Yaskawa INFORM job: DEMO_ROOF_SIDE_0625_3PAINT_61.JBI

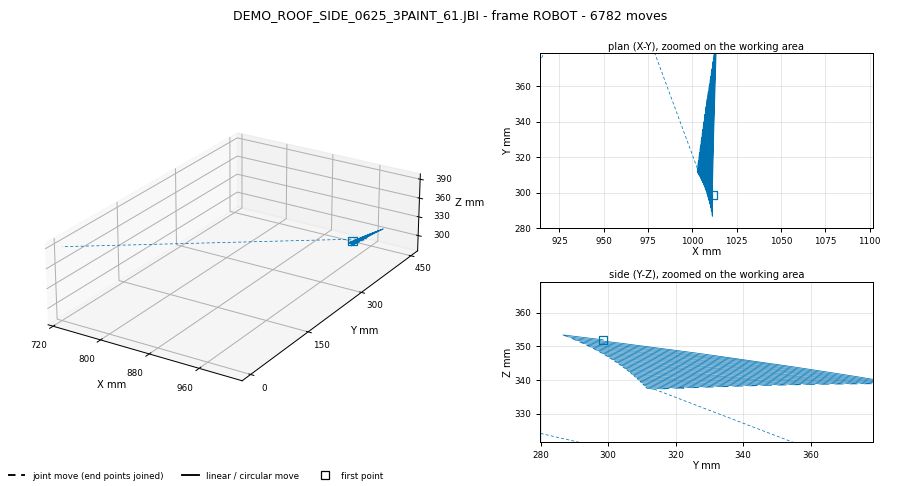
[picture p0: tool path of DEMO_ROOF_SIDE_0625_3PAINT_61.JBI in frame ROBOT, 6782 of 6782 moves have a stored position in this frame; points joined in program order, loops and branches not executed]
/JOB
//NAME DEMO_ROOF_SIDE_0625_3PAINT61
//POS
///NPOS 6782,0,0,0,0,0
///TOOL 0
///USER 0
///POSTYPE ROBOT
///RECTAN
///RCONF 1,0,0,0,0,0,0,0,0,0,0,0,0,0,0,0,0,0,0,0,0,0,0,0
C00000=1011.478,298.564,351.935,169.230,53.497,160.314
C00001=1011.473,298.316,351.966,169.223,53.504,160.314
C00002=1011.467,298.068,351.996,169.218,53.510,160.315
C00003=1011.462,297.820,352.027,169.211,53.517,160.315
C00004=1011.456,297.573,352.058,169.204,53.524,160.315
C00005=1011.451,297.324,352.089,169.198,53.530,160.315
C00006=1011.445,297.077,352.119,169.192,53.537,160.315
C00007=1011.440,296.828,352.150,169.186,53.544,160.316
C00008=1011.434,296.581,352.180,169.180,53.551,160.316
C00009=1011.429,296.332,352.211,169.174,53.558,160.316
C00010=1011.424,296.084,352.241,169.167,53.565,160.316
C00011=1011.418,295.836,352.272,169.161,53.572,160.317
C00012=1011.413,295.588,352.302,169.155,53.578,160.317
C00013=1011.408,295.340,352.333,169.148,53.585,160.317
C00014=1011.402,295.093,352.363,169.142,53.592,160.317
C00015=1011.398,294.844,352.393,169.136,53.599,160.317
C00016=1011.392,294.596,352.424,169.130,53.605,160.318
C00017=1011.387,294.348,352.455,169.123,53.612,160.318
C00018=1011.381,294.100,352.485,169.117,53.620,160.318
C00019=1011.376,293.852,352.515,169.111,53.626,160.319
C00020=1011.369,293.566,352.550,169.104,53.634,160.319
C00021=1011.364,293.280,352.585,169.097,53.642,160.319
C00022=1011.358,292.995,352.620,169.090,53.650,160.319
C00023=1011.352,292.709,352.655,169.082,53.658,160.320
C00024=1011.347,292.461,352.685,169.077,53.665,160.320
C00025=1011.341,292.212,352.715,169.070,53.672,160.320
C00026=1011.336,291.964,352.745,169.065,53.679,160.321
C00027=1011.331,291.716,352.775,169.058,53.686,160.321
C00028=1011.326,291.468,352.806,169.051,53.693,160.321
C00029=1011.320,291.220,352.835,169.046,53.700,160.321
C00030=1011.315,290.971,352.865,169.039,53.707,160.322
C00031=1011.309,290.724,352.895,169.034,53.714,160.322
C00032=1011.304,290.476,352.925,169.027,53.721,160.322
C00033=1011.298,290.227,352.954,169.021,53.728,160.322
C00034=1011.293,289.979,352.985,169.015,53.736,160.323
C00035=1011.288,289.732,353.014,169.009,53.742,160.323
C00036=1011.283,289.483,353.044,169.002,53.750,160.324
C00037=1011.277,289.235,353.074,168.997,53.757,160.324
C00038=1011.272,288.987,353.103,168.990,53.764,160.324
C00039=1011.267,288.739,353.133,168.985,53.771,160.324
C00040=1011.261,288.491,353.163,168.979,53.779,160.325
C00041=1011.256,288.243,353.192,168.972,53.785,160.325
C00042=1011.251,287.995,353.222,168.967,53.793,160.325
C00043=1011.245,287.746,353.251,168.960,53.800,160.326
C00044=1011.240,287.463,353.285,168.953,53.808,160.326
C00045=1011.233,287.181,353.318,168.946,53.816,160.326
C00046=1011.227,286.898,353.352,168.940,53.824,160.327
C00047=1011.221,286.616,353.386,168.933,53.833,160.327
C00048=1010.990,287.953,352.862,168.938,53.865,160.336
C00049=1010.994,288.177,352.835,168.944,53.858,160.335
C00050=1010.999,288.403,352.809,168.949,53.852,160.335
C00051=1011.004,288.627,352.782,168.955,53.845,160.335
C00052=1011.008,288.853,352.755,168.961,53.839,160.335
C00053=1011.014,289.077,352.728,168.965,53.832,160.334
C00054=1011.018,289.303,352.701,168.971,53.826,160.334
C00055=1011.023,289.527,352.674,168.977,53.819,160.334
C00056=1011.027,289.753,352.647,168.983,53.813,160.334
C00057=1011.033,290.001,352.618,168.989,53.806,160.333
C00058=1011.038,290.249,352.588,168.995,53.799,160.333
C00059=1011.043,290.497,352.558,169.001,53.792,160.333
C00060=1011.049,290.745,352.529,169.007,53.785,160.332
C00061=1011.054,290.993,352.499,169.013,53.778,160.332
C00062=1011.060,291.242,352.469,169.020,53.770,160.332
C00063=1011.064,291.489,352.439,169.025,53.764,160.332
C00064=1011.070,291.738,352.409,169.032,53.756,160.331
C00065=1011.075,291.986,352.379,169.038,53.749,160.331
C00066=1011.081,292.233,352.349,169.044,53.743,160.331
C00067=1011.085,292.482,352.319,169.051,53.736,160.331
C00068=1011.091,292.730,352.289,169.056,53.728,160.330
C00069=1011.096,293.018,352.254,169.063,53.720,160.330
C00070=1011.103,293.306,352.219,169.070,53.712,160.330
C00071=1011.110,293.594,352.183,169.078,53.704,160.329
C00072=1011.115,293.882,352.148,169.085,53.696,160.329
C00073=1011.121,294.130,352.118,169.092,53.689,160.329
C00074=1011.126,294.379,352.087,169.097,53.683,160.329
C00075=1011.131,294.627,352.057,169.104,53.676,160.328
C00076=1011.136,294.874,352.027,169.111,53.669,160.328
C00077=1011.141,295.122,351.997,169.117,53.662,160.328
C00078=1011.147,295.371,351.966,169.123,53.655,160.328
C00079=1011.152,295.618,351.936,169.128,53.648,160.327
C00080=1011.157,295.867,351.905,169.135,53.641,160.327
C00081=1011.163,296.115,351.875,169.141,53.635,160.327
C00082=1011.168,296.363,351.844,169.148,53.628,160.327
C00083=1011.174,296.611,351.814,169.154,53.621,160.327
C00084=1011.179,296.859,351.783,169.160,53.614,160.326
C00085=1011.185,297.107,351.752,169.167,53.607,160.326
C00086=1011.189,297.354,351.722,169.172,53.601,160.326
C00087=1011.195,297.603,351.692,169.179,53.594,160.326
C00088=1011.200,297.851,351.661,169.186,53.587,160.326
C00089=1011.205,298.099,351.630,169.192,53.581,160.325
C00090=1011.211,298.347,351.600,169.198,53.574,160.325
C00091=1011.216,298.595,351.569,169.204,53.567,160.325
C00092=1011.222,298.843,351.539,169.211,53.560,160.325
C00093=1011.227,299.091,351.508,169.218,53.554,160.325
C00094=1011.233,299.339,351.477,169.224,53.547,160.324
C00095=1011.238,299.588,351.446,169.230,53.540,160.324
C00096=1011.244,299.835,351.416,169.237,53.534,160.324
C00097=1011.249,300.084,351.385,169.243,53.527,160.324
C00098=1011.255,300.331,351.354,169.250,53.520,160.324
C00099=1011.260,300.580,351.324,169.255,53.514,160.323
C00100=1011.266,300.827,351.293,169.262,53.507,160.323
C00101=1011.271,301.075,351.262,169.269,53.500,160.323
C00102=1011.277,301.323,351.231,169.275,53.494,160.323
C00103=1011.282,301.571,351.200,169.282,53.487,160.323
C00104=1011.288,301.819,351.169,169.287,53.480,160.323
C00105=1011.294,302.067,351.139,169.295,53.474,160.323
C00106=1011.299,302.315,351.108,169.301,53.467,160.322
C00107=1011.304,302.563,351.077,169.307,53.461,160.322
C00108=1011.311,302.811,351.046,169.314,53.454,160.322
C00109=1011.316,303.059,351.015,169.321,53.448,160.322
C00110=1011.322,303.307,350.985,169.327,53.441,160.322
C00111=1011.327,303.555,350.954,169.333,53.434,160.322
C00112=1011.333,303.803,350.923,169.340,53.428,160.322
C00113=1011.338,304.051,350.892,169.346,53.422,160.321
C00114=1011.345,304.299,350.861,169.353,53.415,160.321
C00115=1011.350,304.547,350.829,169.359,53.409,160.321
C00116=1011.356,304.795,350.799,169.366,53.402,160.321
C00117=1011.362,305.043,350.767,169.373,53.395,160.321
C00118=1011.368,305.291,350.736,169.379,53.389,160.321
C00119=1011.373,305.539,350.706,169.386,53.382,160.321
C00120=1011.380,305.787,350.674,169.393,53.376,160.321
C00121=1011.385,306.035,350.643,169.398,53.370,160.320
C00122=1011.391,306.282,350.612,169.405,53.363,160.320
C00123=1011.396,306.531,350.581,169.412,53.356,160.320
C00124=1011.403,306.778,350.550,169.418,53.350,160.320
C00125=1011.408,307.026,350.519,169.425,53.344,160.320
C00126=1011.414,307.274,350.487,169.432,53.337,160.320
C00127=1011.419,307.522,350.456,169.438,53.331,160.320
C00128=1011.425,307.770,350.424,169.445,53.325,160.320
C00129=1011.433,308.076,350.386,169.454,53.316,160.320
C00130=1011.440,308.383,350.348,169.461,53.309,160.320
C00131=1011.448,308.689,350.309,169.470,53.301,160.319
C00132=1011.455,308.995,350.270,169.479,53.293,160.319
C00133=1011.460,309.243,350.238,169.484,53.287,160.319
C00134=1011.465,309.491,350.206,169.491,53.281,160.319
C00135=1011.471,309.739,350.174,169.498,53.275,160.319
C00136=1011.476,309.986,350.142,169.505,53.269,160.319
C00137=1011.482,310.235,350.110,169.511,53.263,160.319
C00138=1011.488,310.481,350.078,169.518,53.256,160.319
C00139=1011.494,310.730,350.046,169.525,53.250,160.319
C00140=1011.498,310.977,350.014,169.531,53.244,160.319
C00141=1011.504,311.226,349.981,169.538,53.238,160.319
C00142=1011.510,311.473,349.950,169.545,53.232,160.319
C00143=1011.516,311.721,349.918,169.551,53.225,160.319
C00144=1011.521,311.969,349.886,169.559,53.219,160.319
C00145=1011.528,312.216,349.853,169.565,53.213,160.319
C00146=1011.533,312.464,349.822,169.572,53.207,160.319
C00147=1011.538,312.713,349.789,169.578,53.201,160.319
C00148=1011.544,312.961,349.757,169.585,53.195,160.319
C00149=1011.550,313.208,349.725,169.592,53.189,160.319
C00150=1011.556,313.456,349.693,169.599,53.183,160.319
C00151=1011.561,313.703,349.661,169.606,53.177,160.319
C00152=1011.567,313.951,349.628,169.612,53.171,160.319
C00153=1011.573,314.199,349.596,169.619,53.165,160.319
C00154=1011.578,314.447,349.564,169.627,53.158,160.319
C00155=1011.584,314.695,349.531,169.633,53.153,160.319
C00156=1011.590,314.943,349.499,169.640,53.146,160.319
C00157=1011.597,315.190,349.466,169.646,53.141,160.319
C00158=1011.601,315.438,349.434,169.653,53.134,160.319
C00159=1011.608,315.686,349.401,169.661,53.128,160.319
C00160=1011.614,315.934,349.369,169.667,53.123,160.319
C00161=1011.620,316.182,349.337,169.674,53.116,160.319
C00162=1011.625,316.429,349.305,169.681,53.110,160.319
C00163=1011.632,316.677,349.272,169.688,53.105,160.319
C00164=1011.637,316.925,349.240,169.695,53.099,160.319
C00165=1011.643,317.173,349.207,169.701,53.093,160.319
C00166=1011.649,317.421,349.175,169.709,53.087,160.319
C00167=1011.655,317.668,349.143,169.716,53.081,160.319
C00168=1011.661,317.916,349.110,169.722,53.076,160.319
C00169=1011.667,318.164,349.078,169.730,53.069,160.319
C00170=1011.673,318.412,349.044,169.737,53.063,160.319
C00171=1011.679,318.659,349.012,169.743,53.057,160.319
C00172=1011.685,318.907,348.980,169.751,53.052,160.319
C00173=1011.691,319.155,348.947,169.758,53.046,160.320
C00174=1011.698,319.403,348.914,169.764,53.040,160.319
C00175=1011.703,319.651,348.882,169.771,53.034,160.319
C00176=1011.709,319.899,348.849,169.779,53.028,160.320
C00177=1011.715,320.146,348.816,169.785,53.023,160.320
C00178=1011.722,320.394,348.783,169.792,53.016,160.320
C00179=1011.728,320.642,348.751,169.800,53.011,160.320
C00180=1011.734,320.889,348.718,169.806,53.005,160.320
C00181=1011.739,321.138,348.685,169.814,53.000,160.320
C00182=1011.746,321.385,348.652,169.821,52.994,160.320
C00183=1011.752,321.633,348.620,169.827,52.988,160.320
C00184=1011.758,321.880,348.587,169.835,52.982,160.320
C00185=1011.765,322.128,348.554,169.842,52.976,160.320
C00186=1011.770,322.376,348.521,169.849,52.971,160.321
C00187=1011.777,322.624,348.488,169.856,52.965,160.321
C00188=1011.783,322.871,348.455,169.864,52.959,160.321
C00189=1011.791,323.183,348.414,169.873,52.952,160.321
C00190=1011.799,323.495,348.373,169.882,52.945,160.321
C00191=1011.807,323.807,348.331,169.891,52.938,160.321
C00192=1011.815,324.119,348.289,169.900,52.931,160.322
C00193=1011.821,324.366,348.257,169.906,52.925,160.321
C00194=1011.827,324.614,348.224,169.914,52.920,160.322
C00195=1011.833,324.862,348.190,169.921,52.914,160.322
C00196=1011.839,325.109,348.158,169.929,52.908,160.322
C00197=1011.847,325.357,348.124,169.936,52.903,160.322
C00198=1011.853,325.604,348.091,169.943,52.897,160.322
C00199=1011.859,325.852,348.057,169.951,52.891,160.322
C00200=1011.864,326.100,348.024,169.957,52.886,160.323
C00201=1011.871,326.347,347.990,169.965,52.881,160.323
C00202=1011.877,326.595,347.957,169.973,52.875,160.323
C00203=1011.883,326.843,347.923,169.979,52.870,160.323
C00204=1011.889,327.090,347.890,169.986,52.864,160.323
C00205=1011.896,327.338,347.855,169.994,52.859,160.324
C00206=1011.901,327.586,347.822,170.001,52.854,160.324
C00207=1011.908,327.833,347.789,170.008,52.848,160.324
C00208=1011.914,328.081,347.754,170.016,52.843,160.324
C00209=1011.920,328.329,347.721,170.023,52.838,160.324
C00210=1011.926,328.576,347.687,170.030,52.832,160.325
C00211=1011.933,328.824,347.653,170.038,52.827,160.325
C00212=1011.939,329.071,347.620,170.046,52.821,160.325
C00213=1011.946,329.319,347.586,170.052,52.816,160.325
C00214=1011.951,329.567,347.552,170.060,52.811,160.325
C00215=1011.958,329.814,347.519,170.068,52.805,160.326
C00216=1011.964,330.062,347.485,170.074,52.800,160.326
C00217=1011.970,330.310,347.450,170.082,52.795,160.326
C00218=1011.977,330.557,347.417,170.090,52.789,160.326
C00219=1011.983,330.804,347.383,170.097,52.784,160.327
C00220=1011.990,331.052,347.348,170.104,52.778,160.327
C00221=1011.996,331.299,347.315,170.112,52.773,160.327
C00222=1012.002,331.548,347.281,170.119,52.768,160.327
C00223=1012.008,331.795,347.247,170.127,52.762,160.327
C00224=1012.016,332.042,347.212,170.134,52.757,160.328
C00225=1012.022,332.290,347.178,170.142,52.752,160.328
C00226=1012.028,332.538,347.144,170.150,52.747,160.328
C00227=1012.034,332.786,347.110,170.156,52.742,160.328
C00228=1012.040,333.033,347.076,170.164,52.736,160.329
C00229=1012.047,333.281,347.041,170.172,52.731,160.329
C00230=1012.053,333.528,347.007,170.180,52.726,160.329
C00231=1012.059,333.776,346.972,170.186,52.721,160.330
C00232=1012.066,334.024,346.937,170.194,52.716,160.330
C00233=1012.072,334.271,346.903,170.202,52.711,160.330
C00234=1012.079,334.519,346.870,170.210,52.705,160.330
C00235=1012.086,334.766,346.834,170.217,52.701,160.331
C00236=1012.092,335.013,346.800,170.225,52.695,160.331
C00237=1012.098,335.261,346.766,170.233,52.691,160.332
C00238=1012.105,335.509,346.731,170.240,52.685,160.332
C00239=1012.111,335.756,346.697,170.248,52.681,160.332
C00240=1012.117,336.003,346.662,170.255,52.675,160.332
C00241=1012.124,336.251,346.627,170.263,52.670,160.333
C00242=1012.130,336.499,346.593,170.271,52.665,160.333
C00243=1012.137,336.746,346.558,170.278,52.661,160.333
C00244=1012.144,336.993,346.524,170.286,52.655,160.334
C00245=1012.150,337.241,346.489,170.294,52.650,160.334
C00246=1012.157,337.489,346.455,170.302,52.645,160.334
C00247=1012.164,337.736,346.420,170.310,52.640,160.335
C00248=1012.170,337.984,346.384,170.316,52.635,160.335
C00249=1012.178,338.291,346.342,170.326,52.629,160.335
C00250=1012.186,338.599,346.298,170.336,52.623,160.336
C00251=1012.194,338.907,346.255,170.346,52.617,160.337
C00252=1012.202,339.213,346.211,170.355,52.611,160.337
C00253=1012.209,339.461,346.176,170.364,52.606,160.337
C00254=1012.216,339.708,346.141,170.371,52.601,160.338
C00255=1012.223,339.956,346.106,170.378,52.596,160.338
C00256=1012.229,340.203,346.070,170.386,52.591,160.338
C00257=1012.235,340.451,346.035,170.395,52.587,160.339
C00258=1012.242,340.699,346.000,170.403,52.582,160.339
C00259=1012.249,340.946,345.965,170.410,52.576,160.340
C00260=1012.255,341.193,345.930,170.418,52.572,160.340
C00261=1012.262,341.441,345.895,170.426,52.567,160.340
C00262=1012.268,341.688,345.859,170.434,52.562,160.341
C00263=1012.275,341.935,345.823,170.442,52.558,160.341
C00264=1012.282,342.182,345.788,170.450,52.553,160.342
C00265=1012.289,342.430,345.753,170.458,52.548,160.342
C00266=1012.296,342.677,345.718,170.465,52.544,160.343
C00267=1012.302,342.925,345.682,170.473,52.539,160.343
C00268=1012.309,343.173,345.647,170.481,52.534,160.344
C00269=1012.316,343.420,345.611,170.490,52.529,160.344
C00270=1012.323,343.667,345.576,170.498,52.525,160.344
C00271=1012.329,343.915,345.540,170.506,52.520,160.345
C00272=1012.336,344.162,345.505,170.514,52.515,160.345
C00273=1012.343,344.409,345.469,170.521,52.511,160.346
C00274=1012.350,344.657,345.434,170.530,52.506,160.346
C00275=1012.356,344.905,345.398,170.538,52.502,160.347
C00276=1012.363,345.151,345.362,170.546,52.497,160.347
C00277=1012.370,345.399,345.327,170.554,52.492,160.348
C00278=1012.378,345.646,345.291,170.562,52.487,160.348
C00279=1012.384,345.894,345.255,170.571,52.483,160.349
C00280=1012.391,346.141,345.219,170.579,52.478,160.349
C00281=1012.397,346.388,345.184,170.587,52.474,160.350
C00282=1012.404,346.636,345.147,170.594,52.469,160.350
C00283=1012.411,346.883,345.112,170.602,52.465,160.351
C00284=1012.417,347.130,345.076,170.611,52.460,160.351
C00285=1012.425,347.378,345.039,170.619,52.456,160.352
C00286=1012.431,347.625,345.004,170.627,52.451,160.352
C00287=1012.438,347.872,344.968,170.635,52.447,160.353
C00288=1012.445,348.120,344.931,170.644,52.443,160.353
C00289=1012.452,348.366,344.895,170.652,52.438,160.354
C00290=1012.459,348.614,344.858,170.661,52.434,160.355
C00291=1012.466,348.862,344.823,170.669,52.429,160.355
C00292=1012.472,349.109,344.787,170.676,52.425,160.356
C00293=1012.480,349.356,344.750,170.684,52.420,160.356
C00294=1012.486,349.603,344.714,170.693,52.416,160.357
C00295=1012.494,349.851,344.678,170.701,52.412,160.357
C00296=1012.500,350.098,344.641,170.710,52.407,160.358
C00297=1012.508,350.345,344.605,170.718,52.403,160.358
C00298=1012.514,350.592,344.569,170.726,52.399,160.359
C00299=1012.522,350.840,344.532,170.735,52.394,160.360
C00300=1012.528,351.087,344.496,170.743,52.390,160.360
C00301=1012.536,351.334,344.460,170.751,52.386,160.361
C00302=1012.543,351.582,344.423,170.760,52.381,160.361
C00303=1012.550,351.828,344.386,170.768,52.377,160.362
C00304=1012.557,352.076,344.350,170.777,52.373,160.362
C00305=1012.564,352.322,344.314,170.785,52.368,160.363
C00306=1012.571,352.570,344.277,170.794,52.364,160.364
C00307=1012.579,352.818,344.241,170.802,52.360,160.364
C00308=1012.586,353.064,344.204,170.810,52.355,160.365
C00309=1012.594,353.369,344.158,170.821,52.351,160.366
C00310=1012.603,353.675,344.113,170.832,52.346,160.367
C00311=1012.612,353.979,344.068,170.842,52.340,160.367
C00312=1012.621,354.284,344.022,170.852,52.335,160.368
C00313=1012.628,354.531,343.985,170.861,52.331,160.369
C00314=1012.634,354.778,343.948,170.869,52.327,160.369
C00315=1012.642,355.025,343.911,170.879,52.322,160.370
C00316=1012.649,355.273,343.875,170.887,52.318,160.371
C00317=1012.657,355.520,343.837,170.896,52.314,160.371
C00318=1012.665,355.767,343.800,170.904,52.310,160.372
C00319=1012.671,356.014,343.764,170.913,52.306,160.373
C00320=1012.678,356.261,343.726,170.922,52.302,160.373
C00321=1012.685,356.508,343.689,170.930,52.298,160.374
C00322=1012.693,356.756,343.652,170.939,52.294,160.375
C00323=1012.700,357.003,343.615,170.948,52.290,160.376
C00324=1012.708,357.250,343.577,170.956,52.286,160.376
C00325=1012.715,357.497,343.540,170.965,52.282,160.377
C00326=1012.723,357.744,343.503,170.973,52.278,160.378
C00327=1012.730,357.992,343.466,170.982,52.274,160.378
C00328=1012.737,358.239,343.429,170.991,52.270,160.379
C00329=1012.744,358.486,343.391,171.000,52.266,160.380
C00330=1012.752,358.733,343.353,171.009,52.262,160.381
C00331=1012.758,358.979,343.316,171.018,52.258,160.381
C00332=1012.766,359.226,343.278,171.026,52.254,160.382
C00333=1012.773,359.473,343.241,171.035,52.251,160.383
C00334=1012.781,359.721,343.203,171.044,52.247,160.384
C00335=1012.788,359.968,343.165,171.053,52.243,160.384
C00336=1012.795,360.215,343.128,171.061,52.239,160.385
C00337=1012.803,360.462,343.089,171.070,52.235,160.386
C00338=1012.810,360.709,343.052,171.080,52.231,160.387
C00339=1012.817,360.956,343.014,171.089,52.227,160.388
C00340=1012.825,361.203,342.976,171.098,52.224,160.389
C00341=1012.832,361.450,342.939,171.106,52.220,160.389
C00342=1012.839,361.697,342.901,171.115,52.216,160.390
C00343=1012.847,361.943,342.863,171.124,52.212,160.391
C00344=1012.855,362.191,342.825,171.134,52.208,160.392
C00345=1012.862,362.438,342.787,171.143,52.205,160.393
C00346=1012.870,362.685,342.749,171.151,52.201,160.393
C00347=1012.877,362.931,342.711,171.160,52.197,160.394
C00348=1012.885,363.179,342.673,171.169,52.194,160.395
C00349=1012.892,363.426,342.635,171.179,52.190,160.396
C00350=1012.900,363.673,342.597,171.188,52.186,160.397
C00351=1012.907,363.919,342.559,171.197,52.183,160.397
C00352=1012.915,364.167,342.520,171.206,52.179,160.398
C00353=1012.923,364.414,342.483,171.216,52.175,160.399
C00354=1012.930,364.660,342.445,171.225,52.172,160.400
C00355=1012.938,364.907,342.406,171.234,52.168,160.401
C00356=1012.946,365.155,342.368,171.243,52.165,160.402
C00357=1012.954,365.402,342.330,171.253,52.161,160.403
C00358=1012.961,365.648,342.292,171.262,52.157,160.404
C00359=1012.969,365.895,342.253,171.271,52.154,160.405
C00360=1012.977,366.142,342.215,171.280,52.151,160.405
C00361=1012.985,366.389,342.176,171.290,52.147,160.406
C00362=1012.993,366.636,342.138,171.299,52.143,160.407
C00363=1013.000,366.883,342.099,171.308,52.140,160.408
C00364=1013.008,367.130,342.060,171.318,52.136,160.409
C00365=1013.015,367.376,342.022,171.327,52.132,160.410
C00366=1013.023,367.624,341.983,171.336,52.129,160.411
C00367=1013.030,367.870,341.945,171.346,52.126,160.412
C00368=1013.039,368.117,341.905,171.355,52.122,160.413
C00369=1013.048,368.429,341.856,171.367,52.118,160.414
C00370=1013.057,368.742,341.807,171.379,52.114,160.415
C00371=1013.067,369.055,341.758,171.390,52.109,160.416
C00372=1013.077,369.367,341.709,171.403,52.105,160.418
C00373=1013.085,369.614,341.669,171.413,52.102,160.419
C00374=1013.093,369.860,341.631,171.422,52.098,160.420
C00375=1013.101,370.107,341.591,171.431,52.095,160.421
C00376=1013.108,370.355,341.552,171.441,52.091,160.422
C00377=1013.117,370.601,341.513,171.450,52.089,160.423
C00378=1013.124,370.848,341.475,171.460,52.085,160.424
C00379=1013.132,371.095,341.435,171.470,52.082,160.425
C00380=1013.140,371.342,341.396,171.479,52.078,160.426
C00381=1013.149,371.588,341.357,171.489,52.075,160.427
C00382=1013.156,371.835,341.317,171.498,52.072,160.428
C00383=1013.164,372.082,341.279,171.508,52.068,160.429
C00384=1013.172,372.329,341.239,171.518,52.066,160.430
C00385=1013.180,372.575,341.199,171.528,52.062,160.431
C00386=1013.189,372.822,341.160,171.537,52.059,160.432
C00387=1013.196,373.069,341.121,171.548,52.056,160.433
C00388=1013.205,373.316,341.082,171.557,52.053,160.434
C00389=1013.212,373.562,341.043,171.567,52.049,160.435
C00390=1013.220,373.809,341.003,171.576,52.046,160.436
C00391=1013.229,374.055,340.963,171.587,52.043,160.438
C00392=1013.237,374.302,340.924,171.596,52.040,160.439
C00393=1013.245,374.549,340.884,171.606,52.037,160.440
C00394=1013.253,374.796,340.845,171.616,52.034,160.441
C00395=1013.262,375.042,340.805,171.626,52.031,160.442
C00396=1013.269,375.289,340.766,171.636,52.028,160.443
C00397=1013.277,375.536,340.726,171.646,52.025,160.444
C00398=1013.285,375.782,340.685,171.655,52.022,160.445
C00399=1013.294,376.030,340.645,171.666,52.019,160.447
C00400=1013.302,376.276,340.605,171.676,52.015,160.448
C00401=1013.310,376.523,340.565,171.686,52.013,160.449
C00402=1013.318,376.769,340.525,171.696,52.009,160.450
C00403=1013.326,377.016,340.485,171.705,52.007,160.451
C00404=1013.334,377.263,340.445,171.716,52.004,160.453
C00405=1013.343,377.508,340.405,171.727,52.001,160.454
C00406=1013.351,377.755,340.365,171.736,51.998,160.455
C00407=1013.359,378.002,340.324,171.746,51.995,160.456
C00408=1013.368,378.249,340.285,171.756,51.992,160.457
C00409=1013.376,378.495,340.244,171.767,51.989,160.458
C00410=1013.384,378.742,340.203,171.777,51.986,160.460
C00411=1013.392,378.988,340.163,171.787,51.984,160.461
C00412=1013.401,379.235,340.123,171.797,51.980,160.462
C00413=1013.409,379.481,340.082,171.808,51.978,160.463
C00414=1013.417,379.728,340.042,171.817,51.975,160.465
C00415=1013.426,379.975,340.002,171.828,51.972,160.466
C00416=1013.434,380.221,339.961,171.839,51.969,160.467
C00417=1013.442,380.468,339.921,171.849,51.967,160.468
C00418=1013.451,380.714,339.880,171.859,51.964,160.470
C00419=1013.459,380.961,339.840,171.870,51.961,160.471
C00420=1013.468,381.207,339.799,171.880,51.958,160.472
C00421=1013.477,381.453,339.759,171.891,51.955,160.473
C00422=1013.485,381.700,339.718,171.901,51.953,160.475
C00423=1013.493,381.947,339.677,171.911,51.950,160.476
C00424=1013.503,382.193,339.637,171.922,51.947,160.477
C00425=1013.511,382.440,339.596,171.933,51.945,160.479
C00426=1013.520,382.687,339.555,171.943,51.942,160.480
C00427=1013.528,382.933,339.515,171.954,51.939,160.481
C00428=1013.537,383.179,339.473,171.964,51.936,160.483
C00429=1013.548,383.480,339.423,171.977,51.934,160.484
C00430=1013.558,383.781,339.373,171.990,51.930,160.486
C00431=1013.569,384.083,339.323,172.003,51.927,160.488
C00432=1013.580,384.384,339.273,172.017,51.924,160.489
C00433=1013.588,384.631,339.232,172.027,51.921,160.491
C00434=1013.597,384.877,339.191,172.037,51.919,160.492
C00435=1013.606,385.124,339.150,172.048,51.916,160.494
C00436=1013.615,385.370,339.108,172.059,51.914,160.495
C00437=1013.623,385.616,339.067,172.070,51.911,160.496
C00438=1013.632,385.863,339.026,172.080,51.908,160.498
C00439=1013.640,386.109,338.984,172.092,51.906,160.499
C00440=1013.649,386.356,338.942,172.103,51.904,160.501
C00441=1013.305,384.294,338.940,171.994,51.982,160.501
C00442=1013.295,384.035,338.983,171.984,51.985,160.499
C00443=1013.286,383.776,339.026,171.972,51.988,160.498
C00444=1013.277,383.517,339.069,171.961,51.991,160.496
C00445=1013.268,383.257,339.113,171.949,51.994,160.495
C00446=1013.259,383.011,339.153,171.939,51.996,160.494
C00447=1013.250,382.764,339.194,171.929,51.999,160.492
C00448=1013.242,382.518,339.235,171.918,52.001,160.491
C00449=1013.233,382.271,339.275,171.907,52.005,160.490
C00450=1013.225,382.025,339.316,171.897,52.007,160.488
C00451=1013.216,381.778,339.357,171.886,52.010,160.487
C00452=1013.208,381.532,339.397,171.875,52.013,160.486
C00453=1013.200,381.285,339.437,171.865,52.015,160.484
C00454=1013.191,381.038,339.478,171.855,52.018,160.483
C00455=1013.182,380.792,339.518,171.844,52.021,160.482
C00456=1013.174,380.545,339.559,171.833,52.024,160.480
C00457=1013.165,380.299,339.600,171.824,52.027,160.479
C00458=1013.157,380.053,339.640,171.813,52.029,160.478
C00459=1013.148,379.806,339.680,171.803,52.032,160.477
C00460=1013.140,379.559,339.721,171.792,52.035,160.475
C00461=1013.132,379.313,339.761,171.783,52.038,160.474
C00462=1013.123,379.066,339.802,171.772,52.041,160.473
C00463=1013.115,378.819,339.842,171.761,52.044,160.472
C00464=1013.107,378.573,339.882,171.751,52.047,160.470
C00465=1013.099,378.326,339.922,171.742,52.050,160.469
C00466=1013.090,378.079,339.963,171.731,52.052,160.468
C00467=1013.082,377.833,340.002,171.721,52.056,160.467
C00468=1013.074,377.587,340.043,171.711,52.059,160.466
C00469=1013.066,377.340,340.083,171.701,52.062,160.465
C00470=1013.058,377.093,340.124,171.690,52.064,160.463
C00471=1013.049,376.847,340.163,171.680,52.067,160.462
C00472=1013.041,376.601,340.203,171.670,52.071,160.461
C00473=1013.034,376.354,340.243,171.661,52.073,160.460
C00474=1013.025,376.107,340.283,171.650,52.077,160.459
C00475=1013.017,375.861,340.323,171.640,52.080,160.457
C00476=1013.009,375.613,340.364,171.631,52.083,160.456
C00477=1013.001,375.367,340.403,171.620,52.086,160.455
C00478=1012.993,375.120,340.443,171.611,52.089,160.454
C00479=1012.985,374.874,340.483,171.600,52.092,160.453
C00480=1012.977,374.627,340.522,171.591,52.095,160.452
C00481=1012.969,374.380,340.561,171.581,52.098,160.451
C00482=1012.961,374.133,340.601,171.570,52.101,160.449
C00483=1012.953,373.887,340.640,171.561,52.104,160.448
C00484=1012.944,373.640,340.680,171.551,52.108,160.447
C00485=1012.936,373.393,340.720,171.541,52.111,160.446
C00486=1012.928,373.147,340.759,171.531,52.114,160.445
C00487=1012.919,372.900,340.798,171.522,52.117,160.444
C00488=1012.912,372.653,340.837,171.512,52.121,160.443
C00489=1012.904,372.406,340.877,171.502,52.124,160.442
C00490=1012.895,372.159,340.916,171.492,52.128,160.441
C00491=1012.888,371.913,340.955,171.483,52.130,160.440
C00492=1012.880,371.666,340.994,171.473,52.134,160.439
C00493=1012.872,371.419,341.034,171.464,52.137,160.438
C00494=1012.864,371.172,341.073,171.453,52.140,160.437
C00495=1012.856,370.926,341.112,171.444,52.144,160.436
C00496=1012.849,370.678,341.151,171.434,52.147,160.435
C00497=1012.840,370.432,341.190,171.425,52.151,160.434
C00498=1012.833,370.185,341.228,171.414,52.154,160.433
C00499=1012.825,369.938,341.268,171.405,52.157,160.432
C00500=1012.817,369.691,341.307,171.396,52.160,160.431
C00501=1012.809,369.445,341.346,171.386,52.164,160.430
C00502=1012.799,369.130,341.396,171.374,52.169,160.429
C00503=1012.789,368.815,341.445,171.362,52.173,160.427
C00504=1012.779,368.500,341.495,171.350,52.177,160.426
C00505=1012.770,368.186,341.545,171.338,52.182,160.425
C00506=1012.762,367.939,341.583,171.328,52.185,160.424
C00507=1012.754,367.692,341.622,171.319,52.188,160.423
C00508=1012.747,367.445,341.661,171.309,52.192,160.422
C00509=1012.739,367.198,341.699,171.300,52.196,160.421
C00510=1012.731,366.951,341.737,171.292,52.199,160.420
C00511=1012.724,366.704,341.777,171.281,52.202,160.419
C00512=1012.717,366.457,341.815,171.272,52.206,160.418
C00513=1012.709,366.211,341.853,171.263,52.209,160.417
C00514=1012.701,365.964,341.892,171.253,52.213,160.416
C00515=1012.693,365.717,341.930,171.244,52.217,160.415
C00516=1012.685,365.470,341.969,171.236,52.221,160.415
C00517=1012.678,365.223,342.006,171.226,52.225,160.414
C00518=1012.670,364.976,342.045,171.217,52.228,160.413
C00519=1012.662,364.729,342.083,171.208,52.232,160.412
C00520=1012.655,364.482,342.120,171.198,52.235,160.411
C00521=1012.647,364.235,342.159,171.189,52.239,160.410
C00522=1012.639,363.988,342.197,171.180,52.242,160.409
C00523=1012.632,363.741,342.235,171.171,52.246,160.408
C00524=1012.624,363.495,342.273,171.161,52.250,160.408
C00525=1012.617,363.247,342.311,171.152,52.254,160.407
C00526=1012.609,363.000,342.349,171.143,52.257,160.406
C00527=1012.602,362.753,342.387,171.134,52.261,160.405
C00528=1012.594,362.507,342.425,171.125,52.265,160.404
C00529=1012.587,362.259,342.463,171.116,52.269,160.403
C00530=1012.579,362.012,342.501,171.107,52.272,160.402
C00531=1012.572,361.765,342.539,171.098,52.276,160.402
C00532=1012.564,361.518,342.576,171.088,52.280,160.401
C00533=1012.557,361.271,342.614,171.080,52.284,160.400
C00534=1012.550,361.024,342.652,171.071,52.288,160.399
C00535=1012.542,360.777,342.689,171.062,52.292,160.399
C00536=1012.535,360.531,342.728,171.053,52.295,160.398
C00537=1012.528,360.283,342.765,171.045,52.300,160.397
C00538=1012.520,360.036,342.803,171.035,52.303,160.396
C00539=1012.513,359.789,342.840,171.026,52.308,160.395
C00540=1012.506,359.542,342.878,171.017,52.311,160.395
C00541=1012.499,359.295,342.915,171.009,52.315,160.394
C00542=1012.491,359.048,342.954,171.000,52.319,160.393
C00543=1012.484,358.801,342.991,170.991,52.323,160.392
C00544=1012.477,358.554,343.029,170.982,52.327,160.392
C00545=1012.469,358.307,343.066,170.973,52.331,160.391
C00546=1012.462,358.059,343.103,170.964,52.335,160.390
C00547=1012.455,357.812,343.141,170.956,52.339,160.389
C00548=1012.448,357.565,343.178,170.947,52.343,160.389
C00549=1012.440,357.318,343.215,170.938,52.347,160.388
C00550=1012.433,357.071,343.253,170.930,52.351,160.387
C00551=1012.426,356.823,343.289,170.921,52.355,160.387
C00552=1012.418,356.576,343.327,170.911,52.359,160.386
C00553=1012.411,356.330,343.363,170.903,52.363,160.385
C00554=1012.404,356.082,343.400,170.894,52.368,160.384
C00555=1012.397,355.835,343.438,170.886,52.372,160.384
C00556=1012.390,355.588,343.475,170.877,52.376,160.383
C00557=1012.382,355.341,343.511,170.869,52.380,160.382
C00558=1012.375,355.094,343.549,170.860,52.384,160.382
C00559=1012.368,354.846,343.585,170.852,52.388,160.381
C00560=1012.360,354.600,343.622,170.843,52.392,160.380
C00561=1012.353,354.352,343.659,170.835,52.396,160.380
C00562=1012.345,354.045,343.705,170.823,52.402,160.379
C00563=1012.336,353.738,343.751,170.812,52.407,160.378
C00564=1012.327,353.430,343.796,170.802,52.412,160.377
C00565=1012.319,353.124,343.842,170.792,52.417,160.376
C00566=1012.311,352.876,343.878,170.783,52.421,160.376
C00567=1012.304,352.630,343.916,170.775,52.425,160.375
C00568=1012.298,352.382,343.952,170.767,52.430,160.375
C00569=1012.290,352.135,343.989,170.758,52.434,160.374
C00570=1012.283,351.888,344.025,170.749,52.438,160.373
C00571=1012.276,351.640,344.061,170.741,52.443,160.373
C00572=1012.269,351.393,344.098,170.733,52.447,160.372
C00573=1012.262,351.146,344.134,170.724,52.451,160.372
C00574=1012.255,350.899,344.170,170.716,52.456,160.371
C00575=1012.248,350.651,344.207,170.708,52.460,160.370
C00576=1012.241,350.404,344.243,170.699,52.464,160.370
C00577=1012.234,350.157,344.279,170.691,52.469,160.369
C00578=1012.227,349.910,344.316,170.682,52.473,160.369
C00579=1012.220,349.662,344.352,170.674,52.478,160.368
C00580=1012.213,349.415,344.388,170.666,52.482,160.368
C00581=1012.206,349.168,344.425,170.658,52.487,160.367
C00582=1012.199,348.921,344.461,170.649,52.491,160.366
C00583=1012.192,348.672,344.497,170.641,52.496,160.366
C00584=1012.186,348.425,344.533,170.632,52.500,160.365
C00585=1012.179,348.179,344.569,170.624,52.505,160.365
C00586=1012.172,347.931,344.606,170.616,52.509,160.364
C00587=1012.165,347.684,344.641,170.608,52.514,160.364
C00588=1012.159,347.436,344.677,170.599,52.518,160.363
C00589=1012.151,347.189,344.713,170.591,52.523,160.363
C00590=1012.144,346.942,344.749,170.583,52.527,160.362
C00591=1012.138,346.695,344.785,170.574,52.532,160.361
C00592=1012.130,346.447,344.821,170.566,52.536,160.361
C00593=1012.124,346.199,344.857,170.558,52.541,160.361
C00594=1012.117,345.953,344.893,170.551,52.546,160.360
C00595=1012.110,345.705,344.928,170.542,52.550,160.360
C00596=1012.104,345.458,344.964,170.534,52.554,160.359
C00597=1012.097,345.210,345.000,170.526,52.559,160.359
C00598=1012.090,344.963,345.035,170.518,52.564,160.358
C00599=1012.083,344.716,345.071,170.510,52.569,160.358
C00600=1012.077,344.468,345.107,170.502,52.574,160.357
C00601=1012.070,344.221,345.142,170.493,52.578,160.357
C00602=1012.063,343.973,345.177,170.485,52.583,160.356
C00603=1012.055,343.726,345.213,170.477,52.587,160.356
C00604=1012.049,343.479,345.249,170.469,52.592,160.355
C00605=1012.043,343.231,345.284,170.462,52.597,160.355
C00606=1012.036,342.984,345.319,170.454,52.601,160.354
C00607=1012.029,342.737,345.354,170.446,52.606,160.354
C00608=1012.023,342.489,345.390,170.438,52.611,160.353
C00609=1012.016,342.242,345.426,170.429,52.616,160.353
C00610=1012.009,341.995,345.461,170.421,52.620,160.353
C00611=1012.003,341.747,345.496,170.413,52.625,160.352
C00612=1011.996,341.500,345.531,170.407,52.630,160.352
C00613=1011.990,341.252,345.567,170.398,52.635,160.352
C00614=1011.983,341.005,345.602,170.390,52.640,160.351
C00615=1011.976,340.758,345.637,170.382,52.645,160.351
C00616=1011.970,340.510,345.672,170.374,52.650,160.350
C00617=1011.963,340.262,345.707,170.366,52.654,160.350
C00618=1011.956,340.015,345.742,170.358,52.660,160.349
C00619=1011.950,339.767,345.778,170.351,52.664,160.349
C00620=1011.943,339.520,345.813,170.343,52.669,160.349
C00621=1011.937,339.272,345.848,170.335,52.674,160.348
C00622=1011.929,338.963,345.891,170.325,52.680,160.348
C00623=1011.920,338.653,345.936,170.316,52.686,160.347
C00624=1011.912,338.343,345.979,170.306,52.692,160.347
C00625=1011.904,338.033,346.022,170.296,52.699,160.346
C00626=1011.898,337.786,346.057,170.288,52.703,160.346
C00627=1011.891,337.538,346.092,170.280,52.709,160.346
C00628=1011.884,337.291,346.127,170.272,52.714,160.345
C00629=1011.878,337.043,346.161,170.266,52.719,160.345
C00630=1011.872,336.796,346.196,170.258,52.724,160.345
C00631=1011.865,336.548,346.230,170.250,52.729,160.344
C00632=1011.859,336.301,346.265,170.242,52.734,160.344
C00633=1011.851,336.053,346.299,170.234,52.739,160.344
C00634=1011.846,335.806,346.333,170.226,52.744,160.343
C00635=1011.839,335.558,346.369,170.219,52.749,160.343
C00636=1011.832,335.310,346.403,170.211,52.754,160.343
C00637=1011.826,335.063,346.437,170.204,52.760,160.342
C00638=1011.820,334.816,346.472,170.195,52.764,160.342
C00639=1011.813,334.568,346.507,170.189,52.769,160.342
C00640=1011.807,334.321,346.541,170.181,52.775,160.342
C00641=1011.801,334.073,346.575,170.173,52.780,160.341
C00642=1011.794,333.825,346.610,170.165,52.785,160.341
C00643=1011.787,333.578,346.644,170.158,52.791,160.341
C00644=1011.781,333.330,346.678,170.151,52.795,160.340
C00645=1011.775,333.083,346.712,170.143,52.801,160.340
C00646=1011.769,332.835,346.746,170.135,52.806,160.340
C00647=1011.763,332.588,346.781,170.128,52.811,160.339
C00648=1011.756,332.340,346.815,170.120,52.816,160.339
C00649=1011.751,332.092,346.849,170.113,52.821,160.339
C00650=1011.744,331.844,346.883,170.105,52.827,160.339
C00651=1011.738,331.597,346.917,170.097,52.832,160.338
C00652=1011.731,331.349,346.951,170.091,52.837,160.338
C00653=1011.725,331.102,346.985,170.083,52.843,160.338
C00654=1011.718,330.855,347.019,170.075,52.848,160.337
C00655=1011.712,330.607,347.053,170.067,52.853,160.337
C00656=1011.706,330.359,347.088,170.061,52.858,160.337
C00657=1011.699,330.112,347.120,170.053,52.864,160.337
C00658=1011.693,329.864,347.155,170.045,52.869,160.337
C00659=1011.687,329.616,347.189,170.038,52.875,160.336
C00660=1011.680,329.369,347.222,170.031,52.880,160.336
C00661=1011.674,329.121,347.256,170.023,52.885,160.336
C00662=1011.668,328.874,347.290,170.016,52.891,160.336
C00663=1011.661,328.626,347.324,170.008,52.896,160.335
C00664=1011.656,328.378,347.357,170.001,52.901,160.335
C00665=1011.649,328.131,347.391,169.994,52.907,160.335
C00666=1011.643,327.882,347.424,169.986,52.913,160.335
C00667=1011.637,327.635,347.458,169.979,52.918,160.335
C00668=1011.630,327.388,347.492,169.972,52.924,160.335
C00669=1011.625,327.140,347.525,169.964,52.929,160.334
C00670=1011.618,326.892,347.560,169.957,52.935,160.334
C00671=1011.612,326.645,347.592,169.950,52.940,160.334
C00672=1011.606,326.397,347.626,169.942,52.945,160.334
C00673=1011.601,326.149,347.660,169.935,52.951,160.334
C00674=1011.594,325.901,347.693,169.929,52.956,160.333
C00675=1011.588,325.654,347.727,169.921,52.962,160.333
C00676=1011.582,325.406,347.760,169.913,52.967,160.333
C00677=1011.576,325.158,347.793,169.906,52.973,160.333
C00678=1011.569,324.911,347.827,169.899,52.979,160.333
C00679=1011.563,324.663,347.860,169.892,52.984,160.332
C00680=1011.556,324.415,347.892,169.885,52.990,160.332
C00681=1011.550,324.168,347.925,169.877,52.996,160.332
C00682=1011.543,323.853,347.967,169.868,53.003,160.332
C00683=1011.535,323.539,348.009,169.859,53.010,160.332
C00684=1011.526,323.226,348.051,169.850,53.017,160.332
C00685=1011.519,322.912,348.092,169.841,53.025,160.332
C00686=1011.513,322.664,348.125,169.833,53.030,160.331
C00687=1011.506,322.417,348.158,169.827,53.036,160.332
C00688=1011.500,322.168,348.191,169.819,53.042,160.331
C00689=1011.494,321.920,348.224,169.812,53.048,160.331
C00690=1011.488,321.672,348.256,169.806,53.053,160.331
C00691=1011.482,321.425,348.289,169.798,53.059,160.331
C00692=1011.475,321.177,348.322,169.791,53.065,160.331
C00693=1011.470,320.929,348.355,169.783,53.071,160.331
C00694=1011.463,320.682,348.388,169.777,53.077,160.331
C00695=1011.457,320.433,348.420,169.770,53.082,160.331
C00696=1011.451,320.186,348.453,169.762,53.088,160.330
C00697=1011.445,319.938,348.485,169.756,53.094,160.331
C00698=1011.439,319.691,348.518,169.749,53.100,160.330
C00699=1011.434,319.443,348.550,169.741,53.106,160.330
C00700=1011.428,319.195,348.583,169.735,53.111,160.330
C00701=1011.421,318.948,348.616,169.727,53.117,160.330
C00702=1011.415,318.699,348.648,169.720,53.123,160.330
C00703=1011.409,318.452,348.681,169.714,53.129,160.330
C00704=1011.403,318.204,348.713,169.707,53.135,160.330
C00705=1011.397,317.956,348.746,169.699,53.141,160.330
C00706=1011.392,317.709,348.778,169.692,53.147,160.330
C00707=1011.386,317.460,348.810,169.686,53.153,160.330
C00708=1011.380,317.213,348.843,169.679,53.159,160.330
C00709=1011.374,316.965,348.875,169.671,53.165,160.330
C00710=1011.368,316.717,348.908,169.665,53.170,160.330
C00711=1011.363,316.469,348.940,169.657,53.176,160.329
C00712=1011.356,316.222,348.973,169.651,53.182,160.330
C00713=1011.350,315.973,349.005,169.644,53.188,160.330
C00714=1011.344,315.726,349.038,169.637,53.194,160.329
C00715=1011.339,315.478,349.069,169.631,53.200,160.330
C00716=1011.333,315.230,349.103,169.624,53.206,160.329
C00717=1011.327,314.982,349.135,169.616,53.213,160.329
C00718=1011.322,314.735,349.166,169.610,53.218,160.330
C00719=1011.315,314.487,349.199,169.603,53.225,160.329
C00720=1011.309,314.239,349.231,169.596,53.231,160.329
C00721=1011.304,313.991,349.263,169.590,53.237,160.329
C00722=1011.298,313.744,349.296,169.582,53.243,160.329
C00723=1011.292,313.495,349.328,169.575,53.249,160.329
C00724=1011.287,313.248,349.360,169.569,53.255,160.329
C00725=1011.281,313.000,349.392,169.562,53.261,160.329
C00726=1011.275,312.753,349.424,169.556,53.267,160.329
C00727=1011.269,312.504,349.456,169.548,53.273,160.329
C00728=1011.265,312.257,349.488,169.541,53.279,160.329
C00729=1011.259,312.008,349.520,169.535,53.285,160.329
C00730=1011.253,311.761,349.552,169.528,53.291,160.329
C00731=1011.247,311.513,349.585,169.521,53.298,160.329
C00732=1011.242,311.266,349.617,169.514,53.303,160.329
C00733=1011.236,311.018,349.649,169.507,53.310,160.329
C00734=1011.231,310.770,349.681,169.501,53.316,160.330
C00735=1011.225,310.522,349.713,169.494,53.322,160.330
C00736=1011.220,310.274,349.745,169.487,53.328,160.329
C00737=1011.214,310.026,349.777,169.481,53.334,160.330
C00738=1011.208,309.778,349.808,169.474,53.341,160.329
C00739=1011.203,309.531,349.840,169.468,53.347,160.330
C00740=1011.198,309.282,349.872,169.461,53.353,160.330
C00741=1011.192,309.035,349.904,169.453,53.359,160.330
C00742=1011.186,308.726,349.944,169.446,53.367,160.330
C00743=1011.178,308.417,349.983,169.437,53.375,160.330
C00744=1011.170,308.109,350.022,169.429,53.383,160.330
C00745=1011.163,307.801,350.060,169.420,53.391,160.330
C00746=1011.157,307.553,350.091,169.415,53.398,160.330
C00747=1011.152,307.305,350.122,169.408,53.404,160.330
C00748=1011.145,307.057,350.153,169.400,53.410,160.330
C00749=1011.140,306.809,350.184,169.395,53.417,160.331
C00750=1011.134,306.561,350.216,169.387,53.423,160.330
C00751=1011.129,306.313,350.247,169.381,53.430,160.331
C00752=1011.123,306.066,350.278,169.375,53.436,160.331
C00753=1011.117,305.817,350.309,169.368,53.442,160.331
C00754=1011.112,305.569,350.340,169.361,53.449,160.331
C00755=1011.106,305.322,350.371,169.355,53.455,160.331
C00756=1011.100,305.073,350.403,169.348,53.462,160.331
C00757=1011.094,304.826,350.434,169.341,53.468,160.331
C00758=1011.089,304.578,350.465,169.335,53.475,160.331
C00759=1011.083,304.330,350.495,169.329,53.482,160.332
C00760=1011.077,304.081,350.526,169.321,53.488,160.332
C00761=1011.071,303.834,350.557,169.316,53.494,160.332
C00762=1011.066,303.586,350.588,169.309,53.501,160.332
C00763=1011.060,303.338,350.619,169.302,53.508,160.332
C00764=1011.055,303.090,350.650,169.296,53.514,160.332
C00765=1011.048,302.842,350.681,169.289,53.521,160.332
C00766=1011.043,302.594,350.712,169.282,53.527,160.332
C00767=1011.037,302.346,350.742,169.276,53.534,160.333
C00768=1011.032,302.098,350.773,169.270,53.541,160.333
C00769=1011.027,301.850,350.804,169.263,53.547,160.333
C00770=1011.021,301.602,350.834,169.257,53.554,160.333
C00771=1011.016,301.354,350.865,169.250,53.560,160.333
C00772=1011.010,301.105,350.896,169.244,53.567,160.333
C00773=1011.004,300.858,350.927,169.238,53.574,160.334
C00774=1010.999,300.610,350.958,169.230,53.580,160.334
C00775=1010.993,300.362,350.988,169.225,53.587,160.334
C00776=1010.988,300.114,351.019,169.218,53.594,160.334
C00777=1010.982,299.866,351.050,169.211,53.601,160.334
C00778=1010.977,299.618,351.081,169.206,53.607,160.334
C00779=1010.971,299.370,351.111,169.199,53.614,160.335
C00780=1010.966,299.121,351.141,169.193,53.621,160.335
C00781=1010.961,298.873,351.172,169.186,53.627,160.335
C00782=1010.955,298.625,351.203,169.179,53.634,160.335
C00783=1010.950,298.377,351.233,169.174,53.640,160.335
C00784=1010.945,298.129,351.264,169.167,53.647,160.335
C00785=1010.939,297.882,351.294,169.160,53.654,160.336
C00786=1010.934,297.633,351.325,169.154,53.661,160.336
C00787=1010.928,297.386,351.356,169.148,53.668,160.336
C00788=1010.923,297.137,351.386,169.142,53.674,160.336
C00789=1010.918,296.890,351.416,169.135,53.681,160.336
C00790=1010.913,296.642,351.447,169.129,53.688,160.337
C00791=1010.908,296.393,351.478,169.123,53.695,160.337
C00792=1010.902,296.146,351.508,169.116,53.702,160.337
C00793=1010.897,295.897,351.538,169.110,53.708,160.337
C00794=1010.891,295.649,351.569,169.104,53.715,160.337
C00795=1010.886,295.401,351.600,169.097,53.722,160.338
C00796=1010.881,295.152,351.629,169.091,53.729,160.338
C00797=1010.876,294.905,351.660,169.085,53.736,160.338
C00798=1010.870,294.657,351.690,169.079,53.742,160.338
C00799=1010.866,294.408,351.720,169.073,53.750,160.339
C00800=1010.860,294.161,351.751,169.066,53.757,160.339
C00801=1010.855,293.912,351.781,169.060,53.763,160.339
C00802=1010.849,293.622,351.816,169.053,53.771,160.339
C00803=1010.843,293.332,351.851,169.046,53.779,160.340
C00804=1010.837,293.042,351.886,169.039,53.787,160.340
C00805=1010.831,292.751,351.922,169.030,53.796,160.340
C00806=1010.826,292.503,351.952,169.025,53.802,160.340
C00807=1010.821,292.255,351.983,169.018,53.810,160.341
C00808=1010.815,292.007,352.013,169.013,53.817,160.341
C00809=1010.810,291.759,352.042,169.006,53.824,160.341
C00810=1010.805,291.511,352.072,168.999,53.830,160.341
C00811=1010.800,291.263,352.103,168.994,53.838,160.342
C00812=1010.795,291.015,352.132,168.987,53.845,160.342
C00813=1010.789,290.766,352.162,168.981,53.852,160.342
C00814=1010.780,290.378,352.208,168.972,53.863,160.343
C00815=1010.772,289.989,352.254,168.962,53.874,160.343
C00816=1010.764,289.601,352.301,168.953,53.885,160.344
C00817=1010.755,289.213,352.347,168.942,53.896,160.344
C00818=1010.521,290.405,351.841,168.947,53.927,160.352
C00819=1010.529,290.748,351.800,168.955,53.917,160.351
C00820=1010.536,291.092,351.759,168.964,53.907,160.351
C00821=1010.543,291.437,351.717,168.972,53.897,160.350
C00822=1010.550,291.780,351.676,168.981,53.887,160.350
C00823=1010.555,292.028,351.646,168.987,53.880,160.350
C00824=1010.561,292.276,351.616,168.993,53.874,160.350
C00825=1010.566,292.525,351.586,168.999,53.866,160.349
C00826=1010.571,292.772,351.556,169.006,53.859,160.349
C00827=1010.577,293.065,351.521,169.013,53.851,160.349
C00828=1010.582,293.358,351.484,169.020,53.843,160.349
C00829=1010.589,293.650,351.449,169.028,53.835,160.348
C00830=1010.595,293.943,351.414,169.035,53.827,160.348
C00831=1010.600,294.191,351.383,169.042,53.820,160.348
C00832=1010.605,294.439,351.352,169.047,53.814,160.348
C00833=1010.610,294.687,351.323,169.054,53.807,160.348
C00834=1010.615,294.935,351.292,169.061,53.800,160.347
C00835=1010.621,295.184,351.262,169.066,53.793,160.347
C00836=1010.626,295.432,351.231,169.073,53.785,160.347
C00837=1010.632,295.679,351.201,169.079,53.778,160.347
C00838=1010.636,295.928,351.171,169.085,53.772,160.346
C00839=1010.642,296.175,351.141,169.092,53.765,160.346
C00840=1010.647,296.423,351.110,169.097,53.758,160.346
C00841=1010.652,296.672,351.080,169.104,53.751,160.346
C00842=1010.658,296.920,351.049,169.111,53.744,160.346
C00843=1010.663,297.168,351.019,169.116,53.738,160.345
C00844=1010.668,297.416,350.988,169.123,53.731,160.345
C00845=1010.673,297.664,350.959,169.130,53.725,160.345
C00846=1010.678,297.912,350.928,169.136,53.718,160.345
C00847=1010.684,298.160,350.897,169.143,53.711,160.345
C00848=1010.689,298.408,350.867,169.148,53.705,160.345
C00849=1010.694,298.656,350.836,169.155,53.698,160.344
C00850=1010.700,298.904,350.806,169.162,53.691,160.344
C00851=1010.705,299.153,350.775,169.168,53.684,160.344
C00852=1010.711,299.400,350.745,169.174,53.677,160.344
C00853=1010.716,299.648,350.714,169.181,53.670,160.344
C00854=1010.722,299.896,350.683,169.187,53.664,160.344
C00855=1010.727,300.144,350.652,169.194,53.657,160.344
C00856=1010.733,300.392,350.622,169.201,53.651,160.343
C00857=1010.738,300.640,350.591,169.206,53.644,160.343
C00858=1010.744,300.888,350.561,169.213,53.637,160.343
C00859=1010.749,301.136,350.530,169.220,53.631,160.343
C00860=1010.754,301.384,350.499,169.226,53.624,160.343
C00861=1010.759,301.632,350.469,169.233,53.617,160.343
C00862=1010.765,301.880,350.438,169.238,53.611,160.342
C00863=1010.771,302.129,350.407,169.245,53.605,160.342
C00864=1010.777,302.377,350.377,169.252,53.598,160.342
C00865=1010.782,302.625,350.346,169.258,53.591,160.342
C00866=1010.788,302.873,350.315,169.265,53.584,160.342
C00867=1010.793,303.120,350.284,169.272,53.578,160.342
C00868=1010.799,303.368,350.253,169.277,53.571,160.342
C00869=1010.804,303.616,350.222,169.284,53.564,160.341
C00870=1010.810,303.865,350.192,169.291,53.558,160.341
C00871=1010.815,304.113,350.161,169.297,53.552,160.341
C00872=1010.822,304.360,350.130,169.304,53.545,160.341
C00873=1010.827,304.608,350.099,169.311,53.538,160.341
C00874=1010.832,304.856,350.068,169.317,53.532,160.341
C00875=1010.838,305.105,350.037,169.324,53.526,160.341
C00876=1010.844,305.352,350.006,169.331,53.519,160.341
C00877=1010.849,305.600,349.975,169.338,53.513,160.341
C00878=1010.855,305.848,349.945,169.344,53.506,160.340
C00879=1010.861,306.096,349.913,169.351,53.500,160.341
C00880=1010.867,306.344,349.882,169.357,53.493,160.340
C00881=1010.872,306.592,349.851,169.364,53.487,160.340
C00882=1010.879,306.840,349.820,169.370,53.480,160.340
C00883=1010.884,307.088,349.789,169.378,53.474,160.340
C00884=1010.890,307.335,349.758,169.383,53.467,160.340
C00885=1010.896,307.584,349.726,169.390,53.461,160.340
C00886=1010.902,307.831,349.695,169.397,53.454,160.340
C00887=1010.909,308.142,349.656,169.406,53.447,160.340
C00888=1010.916,308.453,349.617,169.413,53.439,160.340
C00889=1010.923,308.763,349.578,169.422,53.431,160.340
C00890=1010.930,309.074,349.538,169.430,53.423,160.339
C00891=1010.936,309.323,349.506,169.437,53.416,160.340
C00892=1010.941,309.570,349.474,169.444,53.410,160.339
C00893=1010.947,309.819,349.442,169.451,53.404,160.340
C00894=1010.952,310.066,349.411,169.457,53.397,160.339
C00895=1010.957,310.314,349.379,169.464,53.392,160.339
C00896=1010.963,310.562,349.347,169.471,53.385,160.339
C00897=1010.969,310.809,349.315,169.478,53.379,160.339
C00898=1010.974,311.058,349.283,169.484,53.373,160.339
C00899=1010.979,311.305,349.251,169.491,53.367,160.339
C00900=1010.985,311.553,349.219,169.497,53.361,160.339
C00901=1010.991,311.801,349.187,169.504,53.354,160.339
C00902=1010.996,312.049,349.156,169.512,53.348,160.339
C00903=1011.002,312.297,349.124,169.518,53.342,160.339
C00904=1011.007,312.544,349.091,169.525,53.336,160.339
C00905=1011.013,312.792,349.059,169.532,53.330,160.339
C00906=1011.018,313.040,349.027,169.538,53.324,160.339
C00907=1011.024,313.288,348.995,169.545,53.318,160.339
C00908=1011.030,313.536,348.963,169.553,53.312,160.339
C00909=1011.036,313.783,348.930,169.559,53.306,160.339
C00910=1011.041,314.032,348.898,169.566,53.300,160.339
C00911=1011.047,314.279,348.866,169.572,53.294,160.339
C00912=1011.053,314.527,348.834,169.579,53.288,160.339
C00913=1011.059,314.775,348.801,169.587,53.281,160.339
C00914=1011.064,315.022,348.770,169.593,53.276,160.339
C00915=1011.070,315.271,348.738,169.600,53.269,160.339
C00916=1011.075,315.518,348.705,169.607,53.263,160.339
C00917=1011.081,315.766,348.673,169.613,53.257,160.339
C00918=1011.087,316.014,348.641,169.621,53.251,160.339
C00919=1011.094,316.262,348.608,169.628,53.246,160.340
C00920=1011.099,316.509,348.576,169.635,53.239,160.340
C00921=1011.105,316.757,348.544,169.642,53.234,160.340
C00922=1011.110,317.005,348.511,169.649,53.227,160.340
C00923=1011.117,317.253,348.478,169.656,53.221,160.340
C00924=1011.122,317.501,348.446,169.662,53.215,160.340
C00925=1011.128,317.748,348.414,169.670,53.210,160.340
C00926=1011.134,317.996,348.382,169.677,53.204,160.340
C00927=1011.141,318.244,348.349,169.683,53.198,160.340
C00928=1011.145,318.492,348.317,169.691,53.192,160.340
C00929=1011.152,318.739,348.284,169.698,53.186,160.340
C00930=1011.158,318.987,348.251,169.704,53.180,160.340
C00931=1011.164,319.235,348.219,169.712,53.174,160.340
C00932=1011.170,319.483,348.186,169.719,53.168,160.340
C00933=1011.176,319.731,348.153,169.726,53.162,160.341
C00934=1011.182,319.979,348.121,169.733,53.157,160.341
C00935=1011.188,320.227,348.088,169.740,53.151,160.341
C00936=1011.194,320.474,348.056,169.747,53.145,160.341
C00937=1011.200,320.722,348.024,169.754,53.139,160.341
C00938=1011.206,320.969,347.991,169.761,53.134,160.341
C00939=1011.212,321.217,347.958,169.769,53.127,160.341
C00940=1011.218,321.465,347.925,169.776,53.122,160.341
C00941=1011.224,321.712,347.892,169.782,53.116,160.341
C00942=1011.230,321.961,347.860,169.790,53.110,160.341
C00943=1011.236,322.208,347.828,169.797,53.104,160.342
C00944=1011.243,322.457,347.794,169.804,53.098,160.342
C00945=1011.249,322.704,347.761,169.811,53.093,160.342
C00946=1011.255,322.952,347.728,169.818,53.087,160.342
C00947=1011.263,323.268,347.687,169.828,53.080,160.342
C00948=1011.271,323.584,347.645,169.837,53.073,160.342
C00949=1011.278,323.900,347.603,169.847,53.065,160.342
C00950=1011.287,324.217,347.560,169.856,53.058,160.343
C00951=1011.293,324.465,347.528,169.863,53.052,160.343
C00952=1011.299,324.712,347.495,169.870,53.047,160.343
C00953=1011.306,324.960,347.462,169.877,53.041,160.343
C00954=1011.312,325.208,347.429,169.884,53.035,160.343
C00955=1011.318,325.456,347.396,169.892,53.030,160.343
C00956=1011.324,325.703,347.362,169.899,53.025,160.344
C00957=1011.330,325.951,347.329,169.906,53.019,160.344
C00958=1011.336,326.199,347.296,169.914,53.013,160.344
C00959=1011.342,326.446,347.262,169.921,53.007,160.344
C00960=1011.349,326.694,347.229,169.928,53.002,160.344
C00961=1011.354,326.942,347.194,169.936,52.997,160.345
C00962=1011.361,327.189,347.162,169.943,52.991,160.345
C00963=1011.367,327.437,347.128,169.950,52.986,160.345
C00964=1011.372,327.684,347.094,169.957,52.980,160.345
C00965=1011.379,327.932,347.061,169.965,52.974,160.345
C00966=1011.385,328.180,347.027,169.972,52.969,160.346
C00967=1011.391,328.427,346.993,169.979,52.964,160.346
C00968=1011.398,328.676,346.960,169.987,52.958,160.346
C00969=1011.404,328.923,346.926,169.994,52.953,160.346
C00970=1011.409,329.170,346.892,170.002,52.947,160.346
C00971=1011.416,329.418,346.859,170.009,52.942,160.347
C00972=1011.422,329.666,346.825,170.016,52.937,160.347
C00973=1011.428,329.913,346.791,170.024,52.931,160.347
C00974=1011.435,330.161,346.758,170.032,52.926,160.347
C00975=1011.441,330.409,346.724,170.039,52.920,160.348
C00976=1011.448,330.656,346.690,170.046,52.915,160.348
C00977=1011.454,330.904,346.656,170.054,52.910,160.348
C00978=1011.460,331.152,346.622,170.061,52.904,160.348
C00979=1011.467,331.399,346.588,170.069,52.899,160.349
C00980=1011.472,331.646,346.554,170.077,52.894,160.349
C00981=1011.479,331.894,346.520,170.084,52.889,160.349
C00982=1011.485,332.142,346.486,170.091,52.883,160.349
C00983=1011.491,332.390,346.452,170.099,52.878,160.350
C00984=1011.497,332.637,346.417,170.107,52.872,160.350
C00985=1011.504,332.885,346.384,170.114,52.868,160.350
C00986=1011.510,333.132,346.350,170.122,52.862,160.351
C00987=1011.517,333.380,346.315,170.129,52.857,160.351
C00988=1011.523,333.628,346.281,170.137,52.852,160.351
C00989=1011.529,333.875,346.247,170.145,52.847,160.352
C00990=1011.536,334.123,346.212,170.152,52.842,160.352
C00991=1011.542,334.370,346.178,170.159,52.836,160.352
C00992=1011.548,334.618,346.143,170.167,52.831,160.352
C00993=1011.554,334.866,346.109,170.175,52.826,160.353
C00994=1011.560,335.113,346.075,170.183,52.821,160.353
C00995=1011.568,335.360,346.040,170.190,52.816,160.353
C00996=1011.574,335.608,346.006,170.198,52.810,160.353
C00997=1011.580,335.855,345.972,170.206,52.806,160.354
C00998=1011.587,336.103,345.936,170.213,52.800,160.354
C00999=1011.593,336.351,345.902,170.221,52.795,160.355
C01000=1011.599,336.598,345.868,170.229,52.790,160.355
C01001=1011.606,336.845,345.833,170.236,52.785,160.355
C01002=1011.612,337.093,345.798,170.244,52.780,160.356
C01003=1011.619,337.341,345.763,170.252,52.775,160.356
C01004=1011.625,337.588,345.729,170.260,52.770,160.356
C01005=1011.633,337.835,345.695,170.268,52.765,160.357
C01006=1011.639,338.083,345.660,170.276,52.760,160.357
C01007=1011.647,338.395,345.616,170.286,52.754,160.358
C01008=1011.655,338.707,345.572,170.295,52.748,160.358
C01009=1011.663,339.019,345.528,170.305,52.741,160.359
C01010=1011.671,339.331,345.484,170.315,52.735,160.359
C01011=1011.678,339.578,345.449,170.323,52.730,160.359
C01012=1011.685,339.826,345.415,170.330,52.725,160.360
C01013=1011.691,340.074,345.379,170.338,52.720,160.360
C01014=1011.697,340.321,345.344,170.347,52.715,160.361
C01015=1011.704,340.569,345.309,170.355,52.710,160.361
C01016=1011.711,340.816,345.273,170.362,52.706,160.361
C01017=1011.718,341.063,345.238,170.369,52.701,160.362
C01018=1011.724,341.311,345.203,170.378,52.696,160.362
C01019=1011.730,341.558,345.167,170.386,52.691,160.363
C01020=1011.737,341.806,345.132,170.394,52.686,160.363
C01021=1011.744,342.053,345.097,170.402,52.681,160.364
C01022=1011.751,342.300,345.062,170.410,52.677,160.364
C01023=1011.757,342.548,345.027,170.418,52.672,160.364
C01024=1011.764,342.796,344.991,170.426,52.667,160.365
C01025=1011.770,343.043,344.956,170.433,52.663,160.365
C01026=1011.777,343.290,344.921,170.441,52.658,160.366
C01027=1011.784,343.538,344.886,170.450,52.653,160.366
C01028=1011.790,343.785,344.850,170.458,52.648,160.367
C01029=1011.797,344.033,344.815,170.466,52.643,160.367
C01030=1011.804,344.279,344.779,170.474,52.639,160.368
C01031=1011.810,344.527,344.744,170.482,52.634,160.368
C01032=1011.817,344.775,344.708,170.490,52.629,160.368
C01033=1011.824,345.023,344.673,170.498,52.624,160.369
C01034=1011.831,345.269,344.637,170.507,52.620,160.370
C01035=1011.838,345.517,344.602,170.515,52.615,160.370
C01036=1011.844,345.764,344.566,170.523,52.610,160.371
C01037=1011.851,346.012,344.530,170.531,52.606,160.371
C01038=1011.858,346.259,344.495,170.539,52.601,160.371
C01039=1011.865,346.506,344.458,170.548,52.597,160.372
C01040=1011.871,346.754,344.423,170.555,52.592,160.373
C01041=1011.878,347.001,344.387,170.563,52.587,160.373
C01042=1011.885,347.248,344.350,170.572,52.583,160.374
C01043=1011.891,347.496,344.315,170.580,52.579,160.374
C01044=1011.898,347.742,344.279,170.588,52.574,160.375
C01045=1011.905,347.990,344.242,170.596,52.570,160.375
C01046=1011.912,348.238,344.207,170.604,52.565,160.376
C01047=1011.918,348.485,344.170,170.613,52.561,160.376
C01048=1011.926,348.732,344.134,170.621,52.556,160.377
C01049=1011.932,348.979,344.098,170.629,52.551,160.377
C01050=1011.939,349.226,344.063,170.638,52.547,160.378
C01051=1011.946,349.474,344.026,170.646,52.542,160.378
C01052=1011.953,349.721,343.990,170.654,52.538,160.379
C01053=1011.960,349.969,343.953,170.663,52.534,160.380
C01054=1011.967,350.215,343.917,170.671,52.529,160.380
C01055=1011.974,350.463,343.880,170.680,52.525,160.381
C01056=1011.981,350.710,343.845,170.688,52.520,160.381
C01057=1011.988,350.958,343.808,170.696,52.516,160.382
C01058=1011.995,351.204,343.772,170.705,52.512,160.383
C01059=1012.002,351.452,343.735,170.713,52.507,160.383
C01060=1012.009,351.699,343.699,170.721,52.503,160.384
C01061=1012.016,351.947,343.662,170.730,52.499,160.384
C01062=1012.023,352.193,343.627,170.739,52.494,160.385
C01063=1012.030,352.441,343.590,170.748,52.490,160.386
C01064=1012.038,352.689,343.554,170.756,52.485,160.386
C01065=1012.044,352.936,343.517,170.765,52.481,160.387
C01066=1012.052,353.183,343.480,170.773,52.476,160.387
C01067=1012.060,353.492,343.434,170.783,52.472,160.388
C01068=1012.068,353.802,343.389,170.795,52.466,160.389
C01069=1012.078,354.111,343.342,170.805,52.461,160.390
C01070=1012.087,354.420,343.296,170.816,52.456,160.391
C01071=1012.094,354.667,343.260,170.824,52.452,160.392
C01072=1012.101,354.915,343.223,170.833,52.448,160.392
C01073=1012.108,355.162,343.186,170.842,52.443,160.393
C01074=1012.116,355.409,343.149,170.851,52.439,160.394
C01075=1012.123,355.656,343.112,170.859,52.435,160.394
C01076=1012.130,355.904,343.075,170.868,52.431,160.395
C01077=1012.138,356.151,343.038,170.876,52.426,160.396
C01078=1012.144,356.397,343.001,170.885,52.422,160.396
C01079=1012.151,356.645,342.964,170.893,52.418,160.397
C01080=1012.159,356.892,342.927,170.902,52.414,160.398
C01081=1012.167,357.139,342.890,170.912,52.410,160.398
C01082=1012.173,357.387,342.853,170.920,52.405,160.399
C01083=1012.181,357.634,342.815,170.929,52.402,160.400
C01084=1012.187,357.880,342.778,170.938,52.398,160.401
C01085=1012.195,358.127,342.741,170.946,52.394,160.401
C01086=1012.203,358.374,342.704,170.955,52.390,160.402
C01087=1012.210,358.621,342.666,170.965,52.386,160.403
C01088=1012.217,358.869,342.629,170.973,52.382,160.404
C01089=1012.224,359.116,342.591,170.982,52.377,160.404
C01090=1012.232,359.363,342.554,170.991,52.374,160.405
C01091=1012.239,359.610,342.516,170.999,52.370,160.406
C01092=1012.246,359.857,342.479,171.008,52.366,160.407
C01093=1012.253,360.104,342.441,171.018,52.362,160.407
C01094=1012.261,360.351,342.404,171.027,52.358,160.408
C01095=1012.268,360.598,342.366,171.035,52.354,160.409
C01096=1012.275,360.845,342.328,171.044,52.351,160.410
C01097=1012.282,361.092,342.290,171.053,52.347,160.411
C01098=1012.289,361.340,342.252,171.063,52.343,160.412
C01099=1012.296,361.587,342.215,171.071,52.339,160.412
C01100=1012.304,361.833,342.176,171.080,52.335,160.413
C01101=1012.312,362.081,342.138,171.089,52.331,160.414
C01102=1012.319,362.328,342.100,171.099,52.327,160.415
C01103=1012.326,362.575,342.063,171.108,52.324,160.416
C01104=1012.334,362.822,342.025,171.116,52.319,160.416
C01105=1012.341,363.068,341.987,171.125,52.316,160.417
C01106=1012.349,363.316,341.949,171.135,52.312,160.418
C01107=1012.357,363.563,341.911,171.144,52.309,160.419
C01108=1012.364,363.810,341.873,171.153,52.304,160.420
C01109=1012.371,364.056,341.835,171.163,52.301,160.421
C01110=1012.379,364.304,341.797,171.172,52.297,160.422
C01111=1012.387,364.551,341.759,171.181,52.294,160.422
C01112=1012.394,364.797,341.721,171.191,52.290,160.423
C01113=1012.402,365.045,341.683,171.199,52.286,160.424
C01114=1012.410,365.292,341.644,171.208,52.282,160.425
C01115=1012.417,365.538,341.606,171.218,52.278,160.426
C01116=1012.426,365.785,341.568,171.227,52.275,160.427
C01117=1012.433,366.032,341.530,171.236,52.271,160.428
C01118=1012.440,366.279,341.492,171.246,52.267,160.429
C01119=1012.448,366.526,341.453,171.255,52.264,160.430
C01120=1012.456,366.773,341.415,171.264,52.260,160.430
C01121=1012.464,367.020,341.376,171.274,52.257,160.431
C01122=1012.471,367.267,341.338,171.283,52.253,160.432
C01123=1012.479,367.514,341.299,171.294,52.250,160.433
C01124=1012.487,367.760,341.261,171.302,52.246,160.434
C01125=1012.494,368.008,341.222,171.311,52.243,160.435
C01126=1012.502,368.254,341.183,171.321,52.239,160.436
C01127=1012.511,368.538,341.138,171.332,52.235,160.437
C01128=1012.519,368.823,341.093,171.343,52.231,160.438
C01129=1012.528,369.107,341.048,171.354,52.227,160.440
C01130=1012.537,369.391,341.004,171.365,52.224,160.441
C01131=1012.545,369.639,340.965,171.375,52.220,160.442
C01132=1012.553,369.885,340.926,171.384,52.216,160.443
C01133=1012.560,370.132,340.887,171.394,52.213,160.444
C01134=1012.568,370.379,340.848,171.403,52.209,160.445
C01135=1012.577,370.626,340.809,171.412,52.206,160.446
C01136=1012.583,370.873,340.770,171.423,52.203,160.447
C01137=1012.592,371.119,340.731,171.432,52.199,160.448
C01138=1012.600,371.366,340.692,171.442,52.196,160.449
C01139=1012.607,371.613,340.653,171.452,52.193,160.450
C01140=1012.616,371.859,340.613,171.462,52.189,160.451
C01141=1012.624,372.106,340.575,171.471,52.186,160.452
C01142=1012.632,372.353,340.535,171.481,52.183,160.453
C01143=1012.640,372.600,340.495,171.490,52.180,160.454
C01144=1012.648,372.846,340.457,171.501,52.176,160.455
C01145=1012.655,373.093,340.417,171.511,52.173,160.456
C01146=1012.664,373.340,340.378,171.520,52.170,160.457
C01147=1012.672,373.587,340.339,171.531,52.166,160.459
C01148=1012.680,373.834,340.299,171.539,52.163,160.459
C01149=1012.688,374.081,340.260,171.550,52.160,160.461
C01150=1012.696,374.327,340.221,171.559,52.157,160.462
C01151=1012.704,374.574,340.181,171.570,52.154,160.463
C01152=1012.713,374.821,340.141,171.580,52.150,160.464
C01153=1012.720,375.068,340.102,171.589,52.148,160.465
C01154=1012.729,375.314,340.062,171.600,52.144,160.466
C01155=1012.737,375.561,340.022,171.609,52.141,160.467
C01156=1012.745,375.807,339.982,171.620,52.138,160.469
C01157=1012.753,376.054,339.942,171.630,52.135,160.470
C01158=1012.761,376.301,339.902,171.639,52.132,160.471
C01159=1012.769,376.547,339.862,171.650,52.129,160.472
C01160=1012.777,376.794,339.822,171.660,52.126,160.473
C01161=1012.785,377.041,339.783,171.670,52.123,160.474
C01162=1012.793,377.287,339.742,171.680,52.119,160.476
C01163=1012.801,377.534,339.703,171.690,52.116,160.477
C01164=1012.809,377.780,339.662,171.700,52.114,160.478
C01165=1012.817,378.027,339.622,171.711,52.111,160.479
C01166=1012.825,378.273,339.581,171.721,52.107,160.480
C01167=1012.834,378.520,339.542,171.730,52.105,160.481
C01168=1012.842,378.767,339.501,171.741,52.102,160.483
C01169=1012.850,379.014,339.461,171.752,52.099,160.484
C01170=1012.859,379.260,339.421,171.762,52.096,160.485
C01171=1012.867,379.507,339.380,171.772,52.093,160.487
C01172=1012.875,379.753,339.340,171.782,52.090,160.488
C01173=1012.884,379.999,339.300,171.793,52.087,160.489
C01174=1012.893,380.246,339.259,171.803,52.084,160.490
C01175=1012.901,380.493,339.218,171.814,52.081,160.492
C01176=1012.909,380.739,339.178,171.824,52.079,160.493
C01177=1012.918,380.986,339.138,171.834,52.076,160.494
C01178=1012.926,381.233,339.098,171.845,52.073,160.495
C01179=1012.934,381.479,339.057,171.856,52.070,160.497
C01180=1012.943,381.726,339.016,171.866,52.067,160.498
C01181=1012.951,381.972,338.976,171.876,52.065,160.499
C01182=1012.960,382.218,338.935,171.887,52.062,160.501
C01183=1012.618,380.147,338.926,171.781,52.143,160.501
C01184=1012.610,379.901,338.967,171.770,52.146,160.500
C01185=1012.602,379.655,339.007,171.760,52.149,160.499
C01186=1012.593,379.408,339.047,171.750,52.151,160.497
C01187=1012.585,379.161,339.088,171.740,52.155,160.496
C01188=1012.577,378.915,339.128,171.729,52.157,160.495
C01189=1012.568,378.668,339.167,171.719,52.160,160.494
C01190=1012.560,378.422,339.208,171.708,52.164,160.493
C01191=1012.552,378.175,339.248,171.698,52.166,160.491
C01192=1012.543,377.928,339.288,171.688,52.169,160.490
C01193=1012.535,377.681,339.328,171.678,52.172,160.489
C01194=1012.527,377.435,339.369,171.668,52.175,160.488
C01195=1012.519,377.189,339.408,171.658,52.179,160.487
C01196=1012.511,376.942,339.448,171.647,52.181,160.485
C01197=1012.503,376.695,339.489,171.638,52.184,160.484
C01198=1012.495,376.449,339.528,171.627,52.187,160.483
C01199=1012.487,376.202,339.568,171.617,52.191,160.482
C01200=1012.479,375.956,339.609,171.607,52.193,160.481
C01201=1012.470,375.709,339.648,171.597,52.197,160.479
C01202=1012.463,375.462,339.688,171.587,52.200,160.478
C01203=1012.455,375.215,339.728,171.577,52.203,160.477
C01204=1012.447,374.969,339.767,171.567,52.206,160.476
C01205=1012.439,374.722,339.807,171.557,52.209,160.475
C01206=1012.430,374.475,339.846,171.547,52.212,160.474
C01207=1012.423,374.228,339.886,171.537,52.215,160.472
C01208=1012.414,373.982,339.926,171.528,52.219,160.471
C01209=1012.406,373.735,339.965,171.517,52.222,160.470
C01210=1012.399,373.488,340.004,171.507,52.225,160.469
C01211=1012.390,373.242,340.043,171.497,52.228,160.468
C01212=1012.382,372.995,340.083,171.487,52.232,160.467
C01213=1012.375,372.747,340.122,171.478,52.235,160.466
C01214=1012.366,372.501,340.161,171.468,52.238,160.465
C01215=1012.358,372.254,340.200,171.459,52.242,160.464
C01216=1012.351,372.007,340.239,171.448,52.245,160.463
C01217=1012.342,371.761,340.279,171.439,52.248,160.462
C01218=1012.334,371.514,340.318,171.429,52.252,160.461
C01219=1012.327,371.267,340.357,171.419,52.255,160.459
C01220=1012.319,371.021,340.396,171.410,52.259,160.459
C01221=1012.311,370.774,340.435,171.399,52.262,160.457
C01222=1012.303,370.526,340.474,171.390,52.265,160.456
C01223=1012.295,370.280,340.513,171.380,52.269,160.455
C01224=1012.288,370.035,340.551,171.371,52.272,160.454
C01225=1012.280,369.791,340.590,171.362,52.276,160.453
C01226=1012.272,369.546,340.629,171.351,52.279,160.452
C01227=1012.264,369.301,340.667,171.342,52.282,160.451
C01228=1012.257,369.057,340.706,171.333,52.286,160.451
C01229=1012.249,368.812,340.744,171.323,52.289,160.449
C01230=1012.242,368.568,340.783,171.314,52.293,160.448
C01231=1012.234,368.323,340.821,171.305,52.296,160.448
C01232=1012.226,368.076,340.859,171.295,52.300,160.447
C01233=1012.219,367.829,340.898,171.286,52.303,160.445
C01234=1012.211,367.582,340.937,171.276,52.307,160.444
C01235=1012.203,367.335,340.975,171.267,52.310,160.444
C01236=1012.196,367.088,341.014,171.258,52.314,160.443
C01237=1012.189,366.842,341.052,171.248,52.318,160.442
C01238=1012.181,366.594,341.091,171.239,52.321,160.441
C01239=1012.173,366.348,341.129,171.229,52.325,160.440
C01240=1012.165,366.101,341.168,171.220,52.328,160.439
C01241=1012.157,365.854,341.206,171.211,52.332,160.438
C01242=1012.151,365.607,341.244,171.201,52.336,160.437
C01243=1012.143,365.359,341.283,171.192,52.339,160.436
C01244=1012.135,365.113,341.321,171.182,52.343,160.435
C01245=1012.128,364.866,341.359,171.173,52.347,160.434
C01246=1012.120,364.619,341.397,171.164,52.350,160.433
C01247=1012.112,364.372,341.435,171.154,52.354,160.432
C01248=1012.105,364.125,341.473,171.145,52.358,160.432
C01249=1012.098,363.878,341.511,171.137,52.362,160.431
C01250=1012.090,363.631,341.549,171.127,52.366,160.430
C01251=1012.082,363.384,341.587,171.118,52.369,160.429
C01252=1012.075,363.137,341.625,171.109,52.373,160.428
C01253=1012.067,362.890,341.663,171.100,52.377,160.428
C01254=1012.060,362.643,341.701,171.090,52.381,160.427
C01255=1012.052,362.395,341.738,171.081,52.384,160.426
C01256=1012.045,362.149,341.777,171.073,52.388,160.425
C01257=1012.037,361.902,341.814,171.063,52.392,160.424
C01258=1012.030,361.655,341.852,171.054,52.396,160.423
C01259=1012.023,361.408,341.890,171.045,52.400,160.422
C01260=1012.015,361.161,341.928,171.036,52.403,160.422
C01261=1012.008,360.914,341.965,171.027,52.408,160.421
C01262=1012.001,360.667,342.003,171.018,52.411,160.420
C01263=1011.994,360.420,342.040,171.009,52.415,160.419
C01264=1011.986,360.173,342.078,171.000,52.419,160.418
C01265=1011.979,359.926,342.116,170.991,52.423,160.418
C01266=1011.972,359.679,342.153,170.982,52.428,160.417
C01267=1011.964,359.432,342.191,170.973,52.431,160.416
C01268=1011.957,359.185,342.228,170.965,52.435,160.415
C01269=1011.950,358.937,342.266,170.956,52.439,160.414
C01270=1011.943,358.690,342.304,170.946,52.443,160.414
C01271=1011.935,358.443,342.341,170.937,52.447,160.413
C01272=1011.928,358.196,342.379,170.928,52.451,160.412
C01273=1011.922,357.949,342.415,170.920,52.455,160.411
C01274=1011.914,357.702,342.452,170.911,52.459,160.411
C01275=1011.907,357.455,342.489,170.903,52.463,160.410
C01276=1011.899,357.208,342.527,170.893,52.468,160.409
C01277=1011.892,356.960,342.564,170.884,52.471,160.408
C01278=1011.884,356.713,342.601,170.876,52.475,160.408
C01279=1011.878,356.467,342.638,170.867,52.480,160.407
C01280=1011.871,356.219,342.675,170.859,52.484,160.406
C01281=1011.864,355.972,342.712,170.850,52.488,160.406
C01282=1011.856,355.725,342.748,170.841,52.492,160.405
C01283=1011.849,355.477,342.786,170.832,52.497,160.404
C01284=1011.842,355.230,342.822,170.823,52.501,160.404
C01285=1011.834,354.984,342.859,170.815,52.505,160.403
C01286=1011.827,354.736,342.896,170.806,52.509,160.402
C01287=1011.821,354.489,342.933,170.798,52.513,160.402
C01288=1011.811,354.177,342.980,170.786,52.518,160.401
C01289=1011.803,353.865,343.026,170.776,52.524,160.400
C01290=1011.794,353.553,343.072,170.765,52.529,160.399
C01291=1011.785,353.242,343.118,170.755,52.535,160.398
C01292=1011.778,352.995,343.155,170.746,52.539,160.398
C01293=1011.771,352.748,343.192,170.737,52.543,160.397
C01294=1011.764,352.500,343.228,170.729,52.547,160.396
C01295=1011.757,352.253,343.264,170.720,52.553,160.396
C01296=1011.750,352.006,343.300,170.711,52.557,160.395
C01297=1011.743,351.759,343.337,170.703,52.561,160.394
C01298=1011.736,351.511,343.373,170.694,52.565,160.394
C01299=1011.729,351.264,343.410,170.686,52.570,160.393
C01300=1011.722,351.017,343.446,170.678,52.574,160.393
C01301=1011.715,350.770,343.482,170.669,52.579,160.392
C01302=1011.708,350.522,343.518,170.661,52.583,160.391
C01303=1011.701,350.275,343.555,170.652,52.587,160.391
C01304=1011.694,350.028,343.591,170.644,52.592,160.390
C01305=1011.687,349.781,343.628,170.636,52.596,160.390
C01306=1011.680,349.533,343.663,170.628,52.601,160.389
C01307=1011.674,349.285,343.699,170.619,52.605,160.389
C01308=1011.667,349.039,343.735,170.611,52.610,160.388
C01309=1011.660,348.791,343.772,170.602,52.614,160.387
C01310=1011.653,348.544,343.807,170.594,52.619,160.387
C01311=1011.646,348.297,343.844,170.586,52.623,160.386
C01312=1011.639,348.049,343.880,170.578,52.628,160.386
C01313=1011.633,347.801,343.916,170.569,52.632,160.385
C01314=1011.626,347.555,343.952,170.561,52.637,160.385
C01315=1011.619,347.308,343.988,170.553,52.641,160.384
C01316=1011.612,347.060,344.023,170.544,52.645,160.383
C01317=1011.606,346.813,344.060,170.536,52.650,160.383
C01318=1011.599,346.565,344.095,170.528,52.655,160.383
C01319=1011.593,346.318,344.131,170.520,52.660,160.382
C01320=1011.585,346.070,344.167,170.511,52.664,160.381
C01321=1011.578,345.823,344.203,170.503,52.669,160.381
C01322=1011.572,345.576,344.239,170.495,52.674,160.380
C01323=1011.565,345.328,344.274,170.487,52.678,160.380
C01324=1011.558,345.082,344.310,170.479,52.683,160.380
C01325=1011.551,344.834,344.345,170.470,52.687,160.379
C01326=1011.545,344.586,344.381,170.462,52.692,160.378
C01327=1011.538,344.338,344.416,170.454,52.697,160.378
C01328=1011.531,344.091,344.451,170.446,52.702,160.377
C01329=1011.524,343.844,344.487,170.438,52.707,160.377
C01330=1011.517,343.597,344.522,170.430,52.711,160.377
C01331=1011.511,343.349,344.558,170.422,52.716,160.376
C01332=1011.505,343.102,344.593,170.414,52.721,160.376
C01333=1011.498,342.855,344.628,170.406,52.726,160.375
C01334=1011.491,342.607,344.663,170.398,52.730,160.375
C01335=1011.485,342.359,344.699,170.390,52.735,160.374
C01336=1011.478,342.112,344.734,170.382,52.740,160.374
C01337=1011.472,341.865,344.769,170.374,52.745,160.373
C01338=1011.465,341.617,344.804,170.366,52.750,160.373
C01339=1011.459,341.370,344.840,170.358,52.754,160.372
C01340=1011.452,341.122,344.875,170.350,52.760,160.372
C01341=1011.445,340.875,344.910,170.342,52.765,160.372
C01342=1011.439,340.627,344.945,170.334,52.769,160.371
C01343=1011.432,340.380,344.980,170.326,52.774,160.371
C01344=1011.426,340.133,345.015,170.318,52.779,160.370
C01345=1011.420,339.885,345.050,170.311,52.784,160.370
C01346=1011.413,339.637,345.085,170.303,52.789,160.370
C01347=1011.407,339.390,345.120,170.295,52.794,160.369
C01348=1011.398,339.076,345.164,170.285,52.800,160.369
C01349=1011.390,338.761,345.209,170.275,52.807,160.368
C01350=1011.381,338.447,345.253,170.265,52.813,160.368
C01351=1011.374,338.133,345.297,170.255,52.819,160.367
C01352=1011.367,337.886,345.332,170.247,52.824,160.367
C01353=1011.361,337.638,345.366,170.239,52.830,160.367
C01354=1011.354,337.390,345.402,170.231,52.834,160.366
C01355=1011.348,337.143,345.436,170.224,52.840,160.366
C01356=1011.342,336.895,345.470,170.216,52.845,160.365
C01357=1011.335,336.648,345.505,170.208,52.849,160.365
C01358=1011.328,336.400,345.539,170.201,52.855,160.365
C01359=1011.322,336.153,345.573,170.193,52.860,160.365
C01360=1011.315,335.905,345.608,170.185,52.865,160.364
C01361=1011.309,335.657,345.643,170.177,52.870,160.364
C01362=1011.303,335.410,345.677,170.169,52.875,160.363
C01363=1011.296,335.162,345.711,170.162,52.881,160.363
C01364=1011.290,334.916,345.746,170.155,52.885,160.363
C01365=1011.284,334.668,345.780,170.147,52.891,160.362
C01366=1011.277,334.420,345.815,170.139,52.896,160.362
C01367=1011.271,334.172,345.849,170.131,52.901,160.362
C01368=1011.264,333.925,345.883,170.123,52.906,160.361
C01369=1011.258,333.677,345.917,170.116,52.912,160.361
C01370=1011.252,333.429,345.951,170.109,52.916,160.361
C01371=1011.246,333.182,345.985,170.101,52.922,160.361
C01372=1011.239,332.934,346.020,170.093,52.927,160.360
C01373=1011.234,332.687,346.054,170.086,52.933,160.360
C01374=1011.227,332.439,346.088,170.078,52.938,160.360
C01375=1011.221,332.191,346.122,170.071,52.943,160.359
C01376=1011.215,331.943,346.156,170.063,52.948,160.359
C01377=1011.209,331.696,346.191,170.056,52.954,160.359
C01378=1011.202,331.449,346.224,170.048,52.959,160.359
C01379=1011.196,331.201,346.258,170.040,52.964,160.358
C01380=1011.190,330.954,346.292,170.033,52.969,160.358
C01381=1011.183,330.706,346.326,170.026,52.975,160.358
C01382=1011.177,330.458,346.360,170.018,52.980,160.358
C01383=1011.170,330.211,346.393,170.010,52.986,160.357
C01384=1011.164,329.963,346.427,170.003,52.991,160.357
C01385=1011.159,329.716,346.461,169.996,52.996,160.357
C01386=1011.151,329.468,346.495,169.988,53.002,160.357
C01387=1011.146,329.220,346.528,169.981,53.007,160.356
C01388=1011.140,328.973,346.562,169.973,53.013,160.356
C01389=1011.133,328.724,346.595,169.965,53.018,160.356
C01390=1011.127,328.477,346.629,169.959,53.023,160.356
C01391=1011.121,328.230,346.663,169.951,53.029,160.355
C01392=1011.115,327.982,346.696,169.943,53.034,160.355
C01393=1011.109,327.734,346.730,169.936,53.040,160.355
C01394=1011.102,327.487,346.763,169.929,53.046,160.355
C01395=1011.097,327.239,346.796,169.922,53.051,160.355
C01396=1011.091,326.991,346.831,169.914,53.057,160.354
C01397=1011.084,326.743,346.864,169.906,53.062,160.354
C01398=1011.078,326.496,346.898,169.899,53.068,160.354
C01399=1011.073,326.248,346.931,169.892,53.073,160.354
C01400=1011.066,326.000,346.964,169.885,53.079,160.354
C01401=1011.060,325.753,346.998,169.877,53.085,160.353
C01402=1011.055,325.505,347.031,169.870,53.090,160.353
C01403=1011.049,325.258,347.064,169.863,53.095,160.353
C01404=1011.042,325.009,347.097,169.856,53.101,160.353
C01405=1011.035,324.762,347.130,169.848,53.107,160.353
C01406=1011.030,324.514,347.163,169.840,53.112,160.352
C01407=1011.024,324.266,347.196,169.834,53.118,160.353
C01408=1011.016,323.948,347.238,169.824,53.126,160.352
C01409=1011.008,323.629,347.281,169.815,53.133,160.352
C01410=1010.999,323.311,347.323,169.806,53.140,160.352
C01411=1010.992,322.992,347.365,169.796,53.147,160.352
C01412=1010.985,322.744,347.397,169.790,53.153,160.352
C01413=1010.980,322.496,347.431,169.782,53.159,160.351
C01414=1010.973,322.249,347.463,169.775,53.165,160.351
C01415=1010.967,322.001,347.496,169.767,53.170,160.351
C01416=1010.961,321.753,347.528,169.761,53.176,160.351
C01417=1010.955,321.505,347.561,169.754,53.182,160.351
C01418=1010.949,321.258,347.594,169.746,53.188,160.351
C01419=1010.943,321.010,347.627,169.739,53.194,160.351
C01420=1010.937,320.762,347.659,169.732,53.199,160.351
C01421=1010.931,320.514,347.692,169.725,53.206,160.351
C01422=1010.924,320.267,347.725,169.717,53.211,160.350
C01423=1010.918,320.018,347.757,169.710,53.217,160.350
C01424=1010.913,319.771,347.789,169.704,53.223,160.350
C01425=1010.907,319.524,347.822,169.696,53.229,160.350
C01426=1010.901,319.275,347.854,169.689,53.235,160.350
C01427=1010.895,319.028,347.887,169.682,53.241,160.350
C01428=1010.889,318.780,347.919,169.675,53.246,160.350
C01429=1010.883,318.532,347.952,169.668,53.252,160.350
C01430=1010.878,318.284,347.984,169.661,53.259,160.350
C01431=1010.872,318.037,348.017,169.655,53.264,160.350
C01432=1010.866,317.788,348.049,169.647,53.270,160.349
C01433=1010.859,317.541,348.082,169.640,53.276,160.349
C01434=1010.854,317.293,348.113,169.633,53.282,160.349
C01435=1010.848,317.046,348.146,169.627,53.288,160.349
C01436=1010.842,316.797,348.179,169.619,53.294,160.349
C01437=1010.836,316.550,348.211,169.612,53.300,160.349
C01438=1010.831,316.302,348.243,169.605,53.306,160.349
C01439=1010.825,316.054,348.275,169.598,53.312,160.349
C01440=1010.819,315.806,348.308,169.591,53.318,160.349
C01441=1010.814,315.558,348.340,169.585,53.324,160.349
C01442=1010.808,315.310,348.372,169.578,53.330,160.349
C01443=1010.802,315.063,348.405,169.571,53.336,160.349
C01444=1010.796,314.815,348.436,169.563,53.343,160.349
C01445=1010.790,314.567,348.468,169.557,53.348,160.349
C01446=1010.785,314.319,348.500,169.550,53.355,160.349
C01447=1010.779,314.071,348.533,169.543,53.361,160.349
C01448=1010.774,313.824,348.565,169.537,53.367,160.349
C01449=1010.768,313.576,348.597,169.529,53.373,160.349
C01450=1010.762,313.327,348.629,169.522,53.379,160.349
C01451=1010.757,313.080,348.661,169.516,53.385,160.349
C01452=1010.751,312.832,348.693,169.509,53.391,160.349
C01453=1010.746,312.585,348.726,169.502,53.397,160.349
C01454=1010.740,312.337,348.757,169.495,53.403,160.349
C01455=1010.734,312.089,348.790,169.488,53.409,160.349
C01456=1010.729,311.841,348.821,169.481,53.416,160.349
C01457=1010.723,311.593,348.853,169.475,53.421,160.349
C01458=1010.717,311.346,348.885,169.468,53.428,160.349
C01459=1010.711,311.097,348.917,169.460,53.434,160.349
C01460=1010.707,310.850,348.949,169.455,53.440,160.349
C01461=1010.701,310.602,348.981,169.448,53.447,160.349
C01462=1010.695,310.354,349.013,169.441,53.453,160.349
C01463=1010.690,310.106,349.045,169.434,53.459,160.349
C01464=1010.684,309.858,349.077,169.427,53.465,160.349
C01465=1010.679,309.611,349.108,169.421,53.471,160.349
C01466=1010.674,309.362,349.140,169.414,53.478,160.349
C01467=1010.668,309.114,349.172,169.407,53.484,160.349
C01468=1010.661,308.802,349.212,169.398,53.492,160.349
C01469=1010.655,308.488,349.252,169.390,53.500,160.349
C01470=1010.647,308.176,349.291,169.381,53.508,160.349
C01471=1010.640,307.863,349.330,169.373,53.516,160.349
C01472=1010.634,307.614,349.361,169.367,53.522,160.349
C01473=1010.628,307.367,349.392,169.360,53.529,160.349
C01474=1010.623,307.118,349.423,169.353,53.535,160.349
C01475=1010.617,306.871,349.454,169.347,53.542,160.350
C01476=1010.611,306.623,349.485,169.340,53.548,160.349
C01477=1010.605,306.375,349.516,169.333,53.555,160.350
C01478=1010.600,306.126,349.547,169.327,53.561,160.350
C01479=1010.594,305.879,349.578,169.320,53.568,160.350
C01480=1010.589,305.631,349.609,169.313,53.574,160.350
C01481=1010.582,305.383,349.640,169.306,53.581,160.350
C01482=1010.577,305.135,349.672,169.300,53.587,160.350
C01483=1010.571,304.887,349.702,169.294,53.594,160.350
C01484=1010.566,304.639,349.733,169.286,53.600,160.350
C01485=1010.560,304.391,349.763,169.281,53.606,160.350
C01486=1010.555,304.142,349.795,169.274,53.613,160.351
C01487=1010.548,303.895,349.826,169.267,53.620,160.350
C01488=1010.543,303.647,349.857,169.261,53.626,160.351
C01489=1010.538,303.399,349.887,169.254,53.632,160.351
C01490=1010.532,303.151,349.918,169.247,53.639,160.351
C01491=1010.527,302.903,349.948,169.242,53.646,160.351
C01492=1010.522,302.655,349.979,169.234,53.652,160.351
C01493=1010.516,302.407,350.010,169.228,53.659,160.351
C01494=1010.511,302.159,350.040,169.221,53.666,160.351
C01495=1010.505,301.910,350.072,169.215,53.673,160.352
C01496=1010.499,301.663,350.102,169.208,53.679,160.352
C01497=1010.494,301.415,350.133,169.201,53.686,160.352
C01498=1010.488,301.167,350.163,169.196,53.692,160.352
C01499=1010.483,300.919,350.194,169.189,53.699,160.352
C01500=1010.477,300.671,350.225,169.182,53.705,160.352
C01501=1010.472,300.423,350.256,169.176,53.712,160.352
C01502=1010.466,300.175,350.286,169.169,53.719,160.352
C01503=1010.461,299.927,350.317,169.163,53.726,160.353
C01504=1010.456,299.679,350.347,169.157,53.733,160.353
C01505=1010.450,299.431,350.378,169.150,53.739,160.353
C01506=1010.445,299.184,350.408,169.143,53.746,160.353
C01507=1010.441,298.935,350.438,169.137,53.752,160.353
C01508=1010.435,298.687,350.469,169.131,53.759,160.353
C01509=1010.430,298.439,350.500,169.124,53.766,160.354
C01510=1010.424,298.191,350.530,169.118,53.773,160.354
C01511=1010.419,297.942,350.560,169.112,53.780,160.354
C01512=1010.413,297.694,350.591,169.106,53.786,160.354
C01513=1010.408,297.446,350.622,169.099,53.793,160.354
C01514=1010.402,297.199,350.652,169.093,53.800,160.355
C01515=1010.398,296.950,350.682,169.086,53.806,160.355
C01516=1010.392,296.703,350.712,169.080,53.813,160.355
C01517=1010.387,296.455,350.743,169.073,53.820,160.355
C01518=1010.382,296.206,350.773,169.067,53.827,160.355
C01519=1010.377,295.958,350.804,169.061,53.834,160.355
C01520=1010.371,295.711,350.834,169.054,53.841,160.355
C01521=1010.367,295.462,350.864,169.049,53.848,160.356
C01522=1010.361,295.214,350.894,169.042,53.855,160.356
C01523=1010.356,294.965,350.924,169.035,53.862,160.356
C01524=1010.351,294.718,350.954,169.030,53.868,160.357
C01525=1010.346,294.470,350.985,169.023,53.875,160.357
C01526=1010.340,294.222,351.015,169.016,53.882,160.357
C01527=1010.335,293.973,351.045,169.011,53.889,160.357
C01528=1010.330,293.679,351.081,169.003,53.897,160.357
C01529=1010.324,293.384,351.117,168.995,53.905,160.357
C01530=1010.317,293.089,351.153,168.988,53.913,160.358
C01531=1010.312,292.794,351.189,168.981,53.922,160.358
C01532=1010.305,292.479,351.227,168.973,53.931,160.358
C01533=1010.299,292.164,351.266,168.965,53.940,160.359
C01534=1010.292,291.849,351.303,168.957,53.948,160.359
C01535=1010.286,291.535,351.341,168.949,53.957,160.359
C01536=1010.048,292.611,350.846,168.950,53.989,160.367
C01537=1010.050,292.713,350.834,168.953,53.986,160.367
C01538=1010.058,293.112,350.785,168.964,53.975,160.367
C01539=1010.064,293.410,350.749,168.971,53.967,160.366
C01540=1010.070,293.707,350.713,168.978,53.959,160.366
C01541=1010.077,294.004,350.677,168.986,53.950,160.366
C01542=1010.082,294.252,350.646,168.991,53.943,160.365
C01543=1010.087,294.500,350.617,168.998,53.936,160.365
C01544=1010.092,294.748,350.586,169.005,53.929,160.365
C01545=1010.097,294.997,350.557,169.010,53.923,160.365
C01546=1010.102,295.244,350.526,169.017,53.916,160.365
C01547=1010.107,295.492,350.496,169.024,53.909,160.365
C01548=1010.112,295.741,350.465,169.030,53.902,160.364
C01549=1010.118,295.989,350.436,169.036,53.895,160.364
C01550=1010.122,296.236,350.405,169.043,53.888,160.364
C01551=1010.128,296.485,350.376,169.049,53.882,160.364
C01552=1010.133,296.733,350.345,169.055,53.875,160.364
C01553=1010.139,296.981,350.314,169.062,53.868,160.363
C01554=1010.143,297.229,350.284,169.068,53.861,160.363
C01555=1010.149,297.477,350.254,169.074,53.854,160.363
C01556=1010.154,297.725,350.223,169.081,53.847,160.363
C01557=1010.159,297.974,350.193,169.087,53.841,160.363
C01558=1010.164,298.221,350.163,169.093,53.834,160.362
C01559=1010.169,298.470,350.132,169.101,53.827,160.363
C01560=1010.175,298.718,350.102,169.106,53.821,160.362
C01561=1010.179,298.965,350.071,169.113,53.814,160.362
C01562=1010.185,299.213,350.041,169.120,53.807,160.362
C01563=1010.190,299.461,350.010,169.125,53.800,160.362
C01564=1010.196,299.709,349.980,169.132,53.793,160.362
C01565=1010.201,299.958,349.949,169.139,53.786,160.361
C01566=1010.207,300.206,349.919,169.145,53.781,160.361
C01567=1010.212,300.454,349.888,169.152,53.774,160.361
C01568=1010.218,300.702,349.858,169.158,53.767,160.361
C01569=1010.223,300.950,349.827,169.165,53.760,160.361
C01570=1010.229,301.198,349.797,169.171,53.754,160.361
C01571=1010.234,301.446,349.766,169.178,53.747,160.361
C01572=1010.239,301.694,349.735,169.185,53.740,160.361
C01573=1010.245,301.942,349.704,169.190,53.733,160.360
C01574=1010.250,302.190,349.674,169.197,53.727,160.360
C01575=1010.255,302.438,349.643,169.204,53.720,160.360
C01576=1010.261,302.686,349.613,169.210,53.714,160.360
C01577=1010.266,302.934,349.582,169.217,53.707,160.360
C01578=1010.272,303.182,349.551,169.224,53.700,160.360
C01579=1010.277,303.430,349.520,169.230,53.693,160.360
C01580=1010.283,303.677,349.490,169.237,53.688,160.360
C01581=1010.288,303.926,349.459,169.243,53.681,160.360
C01582=1010.295,304.174,349.428,169.250,53.674,160.359
C01583=1010.300,304.422,349.397,169.256,53.668,160.359
C01584=1010.305,304.670,349.367,169.263,53.661,160.359
C01585=1010.310,304.918,349.336,169.270,53.655,160.359
C01586=1010.317,305.165,349.305,169.276,53.648,160.359
C01587=1010.322,305.414,349.274,169.283,53.642,160.359
C01588=1010.328,305.662,349.243,169.290,53.635,160.359
C01589=1010.333,305.910,349.212,169.297,53.629,160.359
C01590=1010.339,306.157,349.181,169.303,53.622,160.359
C01591=1010.344,306.406,349.150,169.310,53.616,160.359
C01592=1010.350,306.653,349.120,169.316,53.609,160.359
C01593=1010.356,306.902,349.089,169.324,53.603,160.359
C01594=1010.362,307.149,349.058,169.329,53.596,160.358
C01595=1010.367,307.398,349.027,169.337,53.590,160.358
C01596=1010.373,307.645,348.996,169.343,53.583,160.358
C01597=1010.379,307.894,348.964,169.349,53.577,160.358
C01598=1010.386,308.209,348.925,169.359,53.568,160.358
C01599=1010.393,308.524,348.886,169.367,53.561,160.358
C01600=1010.401,308.840,348.846,169.376,53.552,160.358
C01601=1010.407,309.155,348.805,169.384,53.544,160.358
C01602=1010.413,309.402,348.774,169.391,53.539,160.358
C01603=1010.418,309.650,348.742,169.397,53.532,160.358
C01604=1010.424,309.898,348.710,169.404,53.525,160.358
C01605=1010.429,310.146,348.678,169.411,53.520,160.358
C01606=1010.434,310.393,348.646,169.418,53.513,160.358
C01607=1010.440,310.642,348.614,169.425,53.507,160.358
C01608=1010.445,310.889,348.582,169.431,53.501,160.358
C01609=1010.451,311.138,348.551,169.438,53.494,160.358
C01610=1010.456,311.386,348.519,169.445,53.488,160.358
C01611=1010.461,311.633,348.487,169.451,53.482,160.358
C01612=1010.467,311.882,348.455,169.458,53.476,160.358
C01613=1010.472,312.129,348.424,169.466,53.470,160.358
C01614=1010.478,312.377,348.391,169.472,53.464,160.358
C01615=1010.484,312.624,348.359,169.479,53.458,160.358
C01616=1010.489,312.872,348.327,169.486,53.451,160.358
C01617=1010.495,313.120,348.295,169.492,53.446,160.358
C01618=1010.500,313.368,348.263,169.500,53.439,160.358
C01619=1010.506,313.616,348.231,169.507,53.433,160.358
C01620=1010.511,313.863,348.199,169.514,53.427,160.358
C01621=1010.517,314.112,348.167,169.520,53.421,160.358
C01622=1010.523,314.359,348.136,169.527,53.415,160.358
C01623=1010.528,314.607,348.102,169.534,53.409,160.358
C01624=1010.534,314.855,348.070,169.541,53.403,160.358
C01625=1010.540,315.103,348.039,169.548,53.397,160.358
C01626=1010.546,315.351,348.007,169.555,53.390,160.358
C01627=1010.551,315.598,347.974,169.562,53.384,160.358
C01628=1010.557,315.846,347.942,169.568,53.378,160.358
C01629=1010.563,316.095,347.910,169.576,53.372,160.358
C01630=1010.568,316.342,347.878,169.583,53.366,160.358
C01631=1010.574,316.590,347.845,169.589,53.361,160.359
C01632=1010.580,316.838,347.813,169.597,53.354,160.359
C01633=1010.586,317.086,347.782,169.604,53.348,160.359
C01634=1010.592,317.333,347.749,169.611,53.342,160.359
C01635=1010.597,317.582,347.716,169.617,53.336,160.359
C01636=1010.603,317.829,347.684,169.625,53.331,160.359
C01637=1010.609,318.077,347.652,169.632,53.324,160.359
C01638=1010.615,318.324,347.619,169.639,53.318,160.359
C01639=1010.621,318.573,347.587,169.645,53.312,160.359
C01640=1010.626,318.820,347.554,169.653,53.307,160.359
C01641=1010.632,319.068,347.522,169.660,53.301,160.359
C01642=1010.638,319.316,347.489,169.667,53.294,160.359
C01643=1010.644,319.564,347.457,169.674,53.289,160.360
C01644=1010.651,319.811,347.425,169.681,53.283,160.360
C01645=1010.656,320.059,347.393,169.688,53.277,160.360
C01646=1010.662,320.307,347.360,169.696,53.271,160.360
C01647=1010.668,320.554,347.327,169.702,53.266,160.360
C01648=1010.674,320.803,347.295,169.709,53.259,160.360
C01649=1010.680,321.050,347.262,169.717,53.254,160.360
C01650=1010.687,321.298,347.229,169.724,53.248,160.360
C01651=1010.693,321.546,347.197,169.731,53.242,160.360
C01652=1010.698,321.794,347.164,169.738,53.236,160.361
C01653=1010.704,322.041,347.131,169.746,53.231,160.361
C01654=1010.711,322.289,347.098,169.753,53.225,160.361
C01655=1010.717,322.537,347.066,169.761,53.219,160.361
C01656=1010.723,322.785,347.034,169.767,53.213,160.361
C01657=1010.729,323.033,347.000,169.775,53.208,160.361
C01658=1010.736,323.353,346.959,169.783,53.200,160.361
C01659=1010.744,323.674,346.916,169.793,53.193,160.362
C01660=1010.752,323.996,346.873,169.802,53.185,160.362
C01661=1010.761,324.316,346.831,169.812,53.178,160.362
C01662=1010.767,324.564,346.798,169.820,53.172,160.362
C01663=1010.773,324.812,346.765,169.826,53.166,160.362
C01664=1010.779,325.059,346.732,169.834,53.161,160.363
C01665=1010.785,325.307,346.699,169.842,53.155,160.363
C01666=1010.791,325.555,346.666,169.849,53.149,160.363
C01667=1010.797,325.802,346.633,169.855,53.144,160.363
C01668=1010.803,326.050,346.599,169.863,53.138,160.363
C01669=1010.809,326.297,346.566,169.871,53.133,160.364
C01670=1010.816,326.546,346.533,169.878,53.127,160.364
C01671=1010.821,326.793,346.499,169.886,53.121,160.364
C01672=1010.827,327.041,346.465,169.892,53.116,160.364
C01673=1010.833,327.289,346.433,169.900,53.111,160.364
C01674=1010.839,327.536,346.399,169.908,53.105,160.365
C01675=1010.845,327.784,346.365,169.915,53.099,160.365
C01676=1010.852,328.031,346.331,169.922,53.094,160.365
C01677=1010.857,328.279,346.298,169.929,53.089,160.365
C01678=1010.864,328.526,346.265,169.937,53.083,160.366
C01679=1010.870,328.774,346.231,169.944,53.077,160.366
C01680=1010.876,329.022,346.197,169.952,53.072,160.366
C01681=1010.882,329.270,346.164,169.959,53.067,160.366
C01682=1010.888,329.517,346.130,169.966,53.061,160.366
C01683=1010.894,329.766,346.096,169.974,53.056,160.367
C01684=1010.901,330.013,346.063,169.982,53.050,160.367
C01685=1010.907,330.261,346.030,169.990,53.045,160.367
C01686=1010.913,330.509,345.995,169.997,53.040,160.368
C01687=1010.920,330.755,345.962,170.004,53.035,160.368
C01688=1010.925,331.003,345.928,170.012,53.029,160.368
C01689=1010.932,331.251,345.894,170.019,53.024,160.368
C01690=1010.938,331.498,345.860,170.027,53.018,160.369
C01691=1010.945,331.746,345.826,170.035,53.013,160.369
C01692=1010.951,331.994,345.792,170.042,53.007,160.369
C01693=1010.956,332.241,345.758,170.049,53.003,160.369
C01694=1010.963,332.489,345.723,170.057,52.997,160.370
C01695=1010.969,332.736,345.691,170.065,52.992,160.370
C01696=1010.976,332.984,345.656,170.072,52.986,160.370
C01697=1010.981,333.232,345.622,170.081,52.981,160.371
C01698=1010.988,333.480,345.588,170.088,52.976,160.371
C01699=1010.994,333.727,345.554,170.095,52.971,160.371
C01700=1011.001,333.974,345.519,170.102,52.965,160.371
C01701=1011.006,334.222,345.485,170.111,52.960,160.372
C01702=1011.013,334.470,345.450,170.118,52.955,160.372
C01703=1011.019,334.717,345.416,170.126,52.950,160.373
C01704=1011.025,334.965,345.382,170.134,52.944,160.373
C01705=1011.032,335.212,345.348,170.141,52.939,160.373
C01706=1011.038,335.460,345.314,170.149,52.934,160.373
C01707=1011.045,335.707,345.279,170.156,52.929,160.374
C01708=1011.051,335.955,345.245,170.165,52.924,160.374
C01709=1011.057,336.202,345.210,170.172,52.919,160.374
C01710=1011.064,336.450,345.176,170.180,52.914,160.375
C01711=1011.070,336.697,345.141,170.188,52.908,160.375
C01712=1011.076,336.945,345.107,170.196,52.904,160.376
C01713=1011.083,337.193,345.072,170.203,52.898,160.376
C01714=1011.089,337.440,345.037,170.211,52.894,160.376
C01715=1011.096,337.687,345.004,170.218,52.888,160.377
C01716=1011.103,337.935,344.969,170.227,52.883,160.377
C01717=1011.110,338.183,344.934,170.234,52.878,160.377
C01718=1011.117,338.499,344.889,170.244,52.872,160.378
C01719=1011.126,338.816,344.845,170.255,52.866,160.379
C01720=1011.133,339.132,344.800,170.265,52.859,160.379
C01721=1011.142,339.449,344.756,170.275,52.853,160.380
C01722=1011.149,339.696,344.721,170.282,52.847,160.380
C01723=1011.155,339.944,344.686,170.290,52.843,160.380
C01724=1011.160,340.191,344.651,170.298,52.838,160.381
C01725=1011.167,340.439,344.616,170.306,52.833,160.381
C01726=1011.174,340.686,344.581,170.314,52.828,160.382
C01727=1011.180,340.934,344.546,170.322,52.823,160.382
C01728=1011.187,341.181,344.511,170.330,52.818,160.382
C01729=1011.194,341.429,344.476,170.338,52.813,160.383
C01730=1011.200,341.676,344.440,170.346,52.808,160.383
C01731=1011.207,341.924,344.405,170.355,52.803,160.384
C01732=1011.214,342.171,344.370,170.363,52.799,160.384
C01733=1011.220,342.419,344.335,170.371,52.794,160.385
C01734=1011.227,342.666,344.300,170.379,52.789,160.385
C01735=1011.233,342.914,344.264,170.387,52.784,160.386
C01736=1011.240,343.161,344.229,170.394,52.780,160.386
C01737=1011.247,343.408,344.194,170.402,52.775,160.386
C01738=1011.253,343.656,344.158,170.410,52.770,160.387
C01739=1011.259,343.903,344.123,170.418,52.765,160.387
C01740=1011.266,344.151,344.088,170.426,52.760,160.388
C01741=1011.273,344.398,344.052,170.435,52.756,160.388
C01742=1011.280,344.645,344.017,170.443,52.751,160.389
C01743=1011.286,344.893,343.981,170.451,52.746,160.389
C01744=1011.293,345.140,343.946,170.459,52.741,160.390
C01745=1011.300,345.387,343.911,170.467,52.737,160.390
C01746=1011.306,345.635,343.875,170.476,52.732,160.391
C01747=1011.313,345.882,343.839,170.484,52.727,160.391
C01748=1011.320,346.130,343.803,170.492,52.723,160.392
C01749=1011.327,346.377,343.768,170.500,52.718,160.392
C01750=1011.333,346.624,343.732,170.508,52.714,160.393
C01751=1011.340,346.872,343.697,170.517,52.709,160.393
C01752=1011.347,347.119,343.660,170.525,52.704,160.394
C01753=1011.354,347.367,343.625,170.533,52.700,160.395
C01754=1011.360,347.614,343.588,170.541,52.695,160.395
C01755=1011.367,347.861,343.553,170.549,52.690,160.396
C01756=1011.374,348.109,343.516,170.558,52.686,160.396
C01757=1011.381,348.356,343.481,170.566,52.681,160.397
C01758=1011.387,348.603,343.445,170.575,52.677,160.397
C01759=1011.394,348.850,343.409,170.583,52.672,160.398
C01760=1011.401,349.098,343.372,170.591,52.668,160.399
C01761=1011.408,349.345,343.337,170.599,52.663,160.399
C01762=1011.414,349.592,343.301,170.608,52.659,160.400
C01763=1011.422,349.840,343.264,170.617,52.654,160.400
C01764=1011.428,350.087,343.228,170.626,52.650,160.401
C01765=1011.436,350.334,343.192,170.634,52.645,160.401
C01766=1011.442,350.582,343.156,170.642,52.641,160.402
C01767=1011.449,350.829,343.120,170.651,52.637,160.403
C01768=1011.456,351.076,343.083,170.659,52.632,160.403
C01769=1011.463,351.323,343.047,170.667,52.628,160.404
C01770=1011.470,351.571,343.011,170.676,52.624,160.405
C01771=1011.477,351.818,342.975,170.684,52.619,160.405
C01772=1011.484,352.065,342.938,170.693,52.615,160.406
C01773=1011.491,352.312,342.902,170.701,52.610,160.406
C01774=1011.498,352.560,342.865,170.709,52.606,160.407
C01775=1011.505,352.807,342.829,170.719,52.601,160.408
C01776=1011.512,353.054,342.793,170.727,52.597,160.408
C01777=1011.519,353.301,342.755,170.736,52.593,160.409
C01778=1011.528,353.615,342.709,170.746,52.587,160.410
C01779=1011.537,353.929,342.663,170.758,52.582,160.411
C01780=1011.545,354.243,342.616,170.769,52.577,160.412
C01781=1011.554,354.557,342.569,170.779,52.571,160.412
C01782=1011.562,354.804,342.533,170.788,52.567,160.413
C01783=1011.569,355.052,342.495,170.796,52.563,160.414
C01784=1011.576,355.299,342.459,170.806,52.558,160.414
C01785=1011.582,355.546,342.422,170.814,52.554,160.415
C01786=1011.590,355.793,342.385,170.823,52.550,160.416
C01787=1011.597,356.041,342.348,170.831,52.546,160.416
C01788=1011.604,356.287,342.311,170.840,52.541,160.417
C01789=1011.612,356.534,342.274,170.849,52.537,160.418
C01790=1011.619,356.782,342.238,170.859,52.533,160.419
C01791=1011.626,357.029,342.200,170.867,52.529,160.420
C01792=1011.633,357.276,342.164,170.876,52.525,160.420
C01793=1011.641,357.523,342.127,170.884,52.521,160.421
C01794=1011.648,357.770,342.089,170.893,52.517,160.422
C01795=1011.655,358.018,342.052,170.903,52.513,160.423
C01796=1011.662,358.265,342.015,170.911,52.509,160.423
C01797=1011.669,358.512,341.977,170.920,52.505,160.424
C01798=1011.676,358.759,341.940,170.928,52.500,160.425
C01799=1011.683,359.006,341.903,170.937,52.497,160.425
C01800=1011.690,359.253,341.865,170.947,52.492,160.426
C01801=1011.698,359.500,341.828,170.956,52.489,160.427
C01802=1011.705,359.747,341.790,170.964,52.485,160.428
C01803=1011.712,359.994,341.752,170.973,52.481,160.428
C01804=1011.719,360.241,341.715,170.983,52.477,160.429
C01805=1011.727,360.489,341.677,170.991,52.473,160.430
C01806=1011.734,360.736,341.640,171.000,52.469,160.431
C01807=1011.741,360.983,341.602,171.009,52.465,160.432
C01808=1011.749,361.229,341.564,171.019,52.461,160.433
C01809=1011.756,361.476,341.527,171.027,52.457,160.433
